C07263=1105.000,381.902,-90.712,-179.506,16.988,151.525
C07264=1105.007,382.149,-90.748,-179.503,16.992,151.526
C07265=1105.012,382.396,-90.785,-179.501,16.996,151.526
C07266=1105.019,382.643,-90.822,-179.498,17.001,151.527
C07267=1105.028,383.057,-90.883,-179.494,17.008,151.528
C07268=1105.037,383.470,-90.944,-179.490,17.016,151.529
C07269=1105.047,383.884,-91.005,-179.484,17.024,151.530
C07270=1105.056,384.298,-91.066,-179.480,17.032,151.531
C07271=1105.061,384.545,-91.103,-179.478,17.037,151.532
C07272=1105.067,384.792,-91.140,-179.476,17.041,151.532
C07273=1105.073,385.040,-91.177,-179.473,17.046,151.533
C07274=1105.078,385.286,-91.213,-179.470,17.051,151.534
C07275=1105.084,385.533,-91.250,-179.468,17.056,151.534
C07276=1105.090,385.781,-91.287,-179.465,17.060,151.535
C07277=1105.096,386.028,-91.323,-179.462,17.065,151.536
C07278=1105.101,386.274,-91.360,-179.460,17.070,151.536
C07279=1105.106,386.522,-91.397,-179.457,17.075,151.537
C07280=1105.112,386.769,-91.434,-179.454,17.080,151.538
C07281=1105.118,387.016,-91.471,-179.453,17.084,151.538
C07282=1105.124,387.264,-91.508,-179.450,17.089,151.539
C07283=1105.129,387.510,-91.544,-179.447,17.094,151.540
C07284=1105.135,387.758,-91.581,-179.445,17.098,151.540
C07285=1105.141,388.005,-91.618,-179.442,17.104,151.541
C07286=1105.147,388.251,-91.656,-179.440,17.108,151.542
C07287=1105.152,388.499,-91.693,-179.437,17.113,151.543
C07288=1105.158,388.746,-91.730,-179.435,17.118,151.543
C07289=1105.163,388.993,-91.766,-179.432,17.123,151.544
C07290=1105.169,389.240,-91.803,-179.429,17.128,151.545
C07291=1105.175,389.487,-91.840,-179.427,17.133,151.546
C07292=1105.181,389.734,-91.878,-179.424,17.138,151.546
C07293=1105.186,389.981,-91.915,-179.422,17.143,151.547
C07294=1105.192,390.229,-91.952,-179.419,17.148,151.548
C07295=1105.198,390.476,-91.988,-179.417,17.153,151.548
C07296=1105.204,390.722,-92.026,-179.414,17.158,151.549
C07297=1105.210,390.970,-92.063,-179.412,17.164,151.550
C07298=1105.216,391.217,-92.100,-179.409,17.168,151.551
C07299=1105.221,391.463,-92.137,-179.407,17.174,151.552
C07300=1105.226,391.711,-92.174,-179.404,17.179,151.552
C07301=1105.232,391.958,-92.211,-179.402,17.184,151.553
C07302=1105.238,392.205,-92.249,-179.399,17.189,151.554
C07303=1105.244,392.452,-92.286,-179.397,17.194,151.555
C07304=1105.249,392.699,-92.324,-179.394,17.199,151.555
C07305=1105.255,392.946,-92.361,-179.392,17.204,151.556
C07306=1105.261,393.194,-92.398,-179.390,17.210,151.557
C07307=1105.267,393.440,-92.436,-179.387,17.215,151.558
C07308=1105.272,393.688,-92.473,-179.385,17.220,151.559
C07309=1105.278,393.934,-92.511,-179.383,17.225,151.560
C07310=1105.284,394.182,-92.548,-179.380,17.231,151.560
C07311=1105.290,394.428,-92.585,-179.378,17.236,151.561
C07312=1105.295,394.676,-92.622,-179.376,17.241,151.562
C07313=1105.301,394.923,-92.660,-179.373,17.247,151.563
C07314=1105.307,395.170,-92.697,-179.371,17.252,151.564
C07315=1105.313,395.417,-92.735,-179.369,17.257,151.565
C07316=1105.318,395.664,-92.772,-179.366,17.263,151.566
C07317=1105.323,395.911,-92.810,-179.364,17.268,151.567
C07318=1105.329,396.158,-92.848,-179.361,17.274,151.567
C07319=1105.334,396.371,-92.881,-179.359,17.278,151.568
C07320=1105.339,396.584,-92.913,-179.358,17.283,151.569
C07321=1105.344,396.797,-92.945,-179.355,17.288,151.570
C07322=1105.349,397.009,-92.977,-179.354,17.293,151.571
C07323=1105.354,397.223,-93.010,-179.351,17.298,151.571
C07324=1105.359,397.435,-93.042,-179.350,17.302,151.572
C07325=1105.364,397.648,-93.075,-179.348,17.307,151.573
C07326=1105.369,397.861,-93.108,-179.345,17.312,151.574
C07327=1105.375,398.108,-93.145,-179.343,17.317,151.575
C07328=1105.380,398.355,-93.182,-179.341,17.323,151.576
C07329=1105.385,398.602,-93.221,-179.339,17.328,151.577
C07330=1105.391,398.849,-93.259,-179.337,17.334,151.578
C07331=1105.397,399.096,-93.296,-179.334,17.340,151.579
C07332=1105.403,399.344,-93.334,-179.332,17.346,151.580
C07333=1105.408,399.591,-93.372,-179.329,17.351,151.580
C07334=1105.414,399.838,-93.410,-179.327,17.357,151.581
C07335=1105.420,400.085,-93.448,-179.325,17.363,151.582
C07336=1105.425,400.331,-93.486,-179.322,17.369,151.584
C07337=1105.431,400.578,-93.524,-179.320,17.375,151.585
C07338=1105.436,400.825,-93.562,-179.318,17.380,151.585
C07339=1105.442,401.072,-93.600,-179.316,17.386,151.587
C07340=1105.448,401.320,-93.638,-179.313,17.392,151.588
C07341=1105.454,401.567,-93.676,-179.311,17.398,151.589
C07342=1105.460,401.814,-93.713,-179.309,17.404,151.590
C07343=1105.465,402.061,-93.752,-179.307,17.409,151.591
C07344=1105.471,402.308,-93.789,-179.305,17.416,151.592
C07345=1105.476,402.555,-93.828,-179.302,17.422,151.593
C07346=1105.482,402.802,-93.866,-179.300,17.428,151.594
C07347=1105.488,403.049,-93.904,-179.299,17.434,151.595
C07348=1105.493,403.296,-93.942,-179.296,17.440,151.596
C07349=1105.499,403.542,-93.981,-179.294,17.446,151.597
C07350=1105.505,403.790,-94.019,-179.292,17.452,151.598
C07351=1105.511,404.037,-94.058,-179.289,17.458,151.599
C07352=1105.517,404.284,-94.095,-179.287,17.464,151.600
C07353=1105.522,404.531,-94.134,-179.285,17.470,151.601
C07354=1105.528,404.778,-94.172,-179.283,17.476,151.603
C07355=1105.533,405.025,-94.210,-179.281,17.482,151.604
C07356=1105.539,405.272,-94.248,-179.279,17.488,151.605
C07357=1105.545,405.518,-94.287,-179.276,17.495,151.606
C07358=1105.551,405.766,-94.325,-179.274,17.501,151.607
C07359=1105.556,406.013,-94.363,-179.272,17.508,151.608
C07360=1105.562,406.260,-94.402,-179.270,17.514,151.609
C07361=1105.568,406.506,-94.440,-179.268,17.520,151.611
C07362=1105.574,406.754,-94.479,-179.266,17.527,151.612
C07363=1105.579,407.001,-94.517,-179.264,17.532,151.613
C07364=1105.585,407.247,-94.556,-179.261,17.539,151.614
C07365=1105.591,407.495,-94.594,-179.259,17.545,151.615
C07366=1105.596,407.742,-94.633,-179.258,17.552,151.617
C07367=1105.602,407.988,-94.671,-179.255,17.558,151.618
C07368=1105.607,408.235,-94.710,-179.254,17.565,151.619
C07369=1105.613,408.483,-94.748,-179.251,17.572,151.620
C07370=1105.618,408.729,-94.787,-179.249,17.578,151.621
C07371=1105.624,408.976,-94.826,-179.247,17.584,151.623
C07372=1105.630,409.223,-94.865,-179.245,17.591,151.624
C07373=1105.636,409.470,-94.903,-179.243,17.598,151.625
C07374=1105.641,409.716,-94.942,-179.241,17.604,151.626
C07375=1105.646,409.930,-94.975,-179.239,17.610,151.628
C07376=1105.650,410.142,-95.008,-179.237,17.616,151.629
C07377=1105.656,410.355,-95.042,-179.235,17.622,151.630
C07378=1105.661,410.568,-95.076,-179.234,17.627,151.631
C07379=1105.665,410.780,-95.109,-179.232,17.633,151.632
C07380=1105.670,410.994,-95.143,-179.230,17.639,151.633
C07381=1105.675,411.206,-95.176,-179.229,17.645,151.634
C07382=1105.680,411.419,-95.209,-179.227,17.651,151.635
C07383=1105.686,411.665,-95.248,-179.225,17.657,151.637
C07384=1105.692,411.913,-95.287,-179.223,17.664,151.638
C07385=1105.697,412.159,-95.326,-179.221,17.671,151.639
C07386=1105.703,412.406,-95.365,-179.219,17.678,151.641
C07387=1105.709,412.653,-95.404,-179.217,17.685,151.642
C07388=1105.714,412.900,-95.443,-179.215,17.692,151.643
C07389=1105.720,413.147,-95.482,-179.213,17.699,151.645
C07390=1105.725,413.394,-95.520,-179.210,17.706,151.646
C07391=1105.731,413.641,-95.560,-179.209,17.713,151.647
C07392=1105.737,413.888,-95.599,-179.207,17.720,151.649
C07393=1105.742,414.134,-95.638,-179.205,17.726,151.650
C07394=1105.748,414.381,-95.677,-179.203,17.734,151.652
C07395=1105.754,414.628,-95.715,-179.201,17.741,151.653
C07396=1105.760,414.875,-95.755,-179.199,17.748,151.654
C07397=1105.766,415.121,-95.794,-179.197,17.755,151.656
C07398=1105.772,415.369,-95.833,-179.195,17.762,151.657
C07399=1105.777,415.615,-95.872,-179.193,17.770,151.659
C07400=1105.783,415.862,-95.912,-179.192,17.776,151.660
C07401=1105.789,416.109,-95.951,-179.189,17.784,151.662
C07402=1105.795,416.356,-95.990,-179.187,17.791,151.663
C07403=1105.800,416.602,-96.029,-179.185,17.799,151.665
C07404=1105.806,416.850,-96.069,-179.184,17.805,151.666
C07405=1105.811,417.096,-96.108,-179.182,17.813,151.667
C07406=1105.817,417.343,-96.148,-179.180,17.820,151.669
C07407=1105.823,417.590,-96.187,-179.178,17.828,151.671
C07408=1105.829,417.837,-96.226,-179.176,17.835,151.672
C07409=1105.834,418.083,-96.265,-179.175,17.843,151.674
C07410=1105.840,418.331,-96.305,-179.173,17.850,151.675
C07411=1105.845,418.577,-96.344,-179.171,17.858,151.677
C07412=1105.851,418.824,-96.384,-179.169,17.865,151.678
C07413=1105.857,419.071,-96.423,-179.167,17.873,151.680
C07414=1105.863,419.318,-96.462,-179.165,17.881,151.681
C07415=1105.868,419.564,-96.503,-179.164,17.888,151.683
C07416=1105.874,419.811,-96.542,-179.162,17.895,151.684
C07417=1105.880,420.058,-96.581,-179.160,17.903,151.686
C07418=1105.885,420.305,-96.621,-179.158,17.911,151.688
C07419=1105.891,420.551,-96.661,-179.156,17.919,151.689
C07420=1105.897,420.798,-96.700,-179.154,17.927,151.691
C07421=1105.903,421.045,-96.740,-179.152,17.934,151.693
C07422=1105.907,421.292,-96.779,-179.151,17.942,151.694
C07423=1105.914,421.538,-96.820,-179.149,17.950,151.696
C07424=1105.920,421.785,-96.859,-179.147,17.958,151.698
C07425=1105.926,422.031,-96.899,-179.146,17.965,151.699
C07426=1105.931,422.279,-96.939,-179.144,17.973,151.701
C07427=1105.937,422.526,-96.978,-179.143,17.982,151.703
C07428=1105.943,422.772,-97.018,-179.141,17.989,151.704
C07429=1105.948,423.019,-97.058,-179.139,17.997,151.706
C07430=1105.954,423.265,-97.098,-179.137,18.005,151.708
C07431=1105.958,423.484,-97.133,-179.135,18.013,151.709
C07432=1105.964,423.704,-97.168,-179.134,18.020,151.711
C07433=1105.969,423.923,-97.205,-179.133,18.027,151.712
C07434=1105.974,424.143,-97.240,-179.131,18.035,151.714
C07435=1105.979,424.362,-97.275,-179.130,18.042,151.715
C07436=1105.984,424.581,-97.311,-179.128,18.050,151.717
C07437=1105.989,424.800,-97.346,-179.127,18.057,151.719
C07438=1105.994,425.020,-97.381,-179.126,18.064,151.720
C07439=1106.000,425.267,-97.422,-179.124,18.072,151.722
C07440=1106.005,425.512,-97.462,-179.122,18.080,151.724
C07441=1106.011,425.760,-97.502,-179.121,18.088,151.725
C07442=1106.017,426.006,-97.542,-179.119,18.098,151.727
C07443=1106.022,426.252,-97.582,-179.117,18.106,151.729
C07444=1106.028,426.500,-97.622,-179.115,18.114,151.731
C07445=1106.034,426.746,-97.663,-179.114,18.123,151.733
C07446=1106.040,426.993,-97.703,-179.112,18.131,151.735
C07447=1106.045,427.239,-97.743,-179.111,18.139,151.737
C07448=1106.051,427.486,-97.783,-179.110,18.148,151.738
C07449=1106.057,427.733,-97.823,-179.108,18.156,151.740
C07450=1106.062,427.979,-97.864,-179.106,18.165,151.742
C07451=1106.068,428.226,-97.904,-179.104,18.174,151.744
C07452=1106.074,428.472,-97.944,-179.103,18.183,151.746
C07453=1106.079,428.720,-97.985,-179.102,18.191,151.748
C07454=1106.085,428.966,-98.024,-179.100,18.200,151.750
C07455=1106.091,429.213,-98.065,-179.099,18.209,151.752
C07456=1106.097,429.459,-98.106,-179.097,18.218,151.754
C07457=1106.103,429.706,-98.146,-179.096,18.226,151.756
C07458=1106.108,429.952,-98.186,-179.094,18.235,151.758
C07459=1106.114,430.199,-98.227,-179.093,18.244,151.760
C07460=1106.120,430.445,-98.267,-179.091,18.254,151.762
C07461=1106.125,430.691,-98.308,-179.090,18.262,151.764
C07462=1106.131,430.938,-98.348,-179.089,18.271,151.766
C07463=1106.136,431.185,-98.389,-179.088,18.280,151.768
C07464=1106.142,431.432,-98.430,-179.086,18.290,151.770
C07465=1106.148,431.678,-98.470,-179.084,18.298,151.772
C07466=1106.153,431.925,-98.510,-179.083,18.308,151.774
C07467=1106.159,432.171,-98.551,-179.081,18.317,151.776
C07468=1106.165,432.418,-98.593,-179.080,18.326,151.778
C07469=1106.171,432.664,-98.633,-179.079,18.335,151.780
C07470=1106.177,432.911,-98.673,-179.077,18.345,151.782
C07471=1106.182,433.157,-98.714,-179.076,18.354,151.784
C07472=1106.188,433.404,-98.755,-179.075,18.363,151.787
C07473=1106.194,433.650,-98.796,-179.073,18.373,151.789
C07474=1106.199,433.897,-98.837,-179.072,18.382,151.791
C07475=1106.205,434.144,-98.877,-179.071,18.391,151.793
C07476=1106.210,434.390,-98.918,-179.070,18.401,151.795
C07477=1106.216,434.636,-98.959,-179.069,18.410,151.797
C07478=1106.222,434.883,-99.000,-179.067,18.421,151.800
C07479=1106.227,435.130,-99.041,-179.066,18.430,151.802
C07480=1106.233,435.376,-99.082,-179.065,18.439,151.804
C07481=1106.238,435.622,-99.123,-179.064,18.449,151.806
C07482=1106.244,435.868,-99.164,-179.063,18.459,151.809
C07483=1106.250,436.115,-99.205,-179.061,18.469,151.811
C07484=1106.255,436.362,-99.246,-179.060,18.478,151.813
C07485=1106.261,436.608,-99.287,-179.059,18.488,151.815
C07486=1106.267,436.855,-99.328,-179.058,18.498,151.818
C07487=1106.272,437.072,-99.364,-179.057,18.507,151.820
C07488=1106.277,437.290,-99.400,-179.056,18.516,151.822
C07489=1106.282,437.508,-99.437,-179.055,18.524,151.824
C07490=1106.287,437.726,-99.474,-179.054,18.533,151.826
C07491=1106.292,437.944,-99.510,-179.053,18.542,151.828
C07492=1106.297,438.162,-99.546,-179.052,18.551,151.830
C07493=1106.302,438.380,-99.582,-179.051,18.560,151.832
C07494=1106.307,438.598,-99.619,-179.050,18.569,151.834
C07495=1106.313,438.844,-99.660,-179.049,18.579,151.837
C07496=1106.318,439.091,-99.701,-179.048,18.589,151.839
C07497=1106.324,439.337,-99.743,-179.047,18.600,151.842
C07498=1106.330,439.583,-99.784,-179.046,18.609,151.844
C07499=1106.336,439.829,-99.825,-179.045,18.620,151.846
C07500=1106.341,440.076,-99.867,-179.044,18.630,151.849
C07501=1106.347,440.323,-99.908,-179.043,18.641,151.851
C07502=1106.353,440.569,-99.950,-179.041,18.651,151.854
C07503=1106.359,440.815,-99.991,-179.041,18.661,151.856
C07504=1106.365,441.062,-100.032,-179.040,18.672,151.859
C07505=1106.370,441.308,-100.074,-179.039,18.682,151.861
C07506=1106.376,441.555,-100.115,-179.038,18.693,151.864
C07507=1106.382,441.801,-100.157,-179.037,18.704,151.866
C07508=1106.388,442.047,-100.198,-179.037,18.714,151.869
C07509=1106.393,442.293,-100.240,-179.036,18.725,151.872
C07510=1106.399,442.540,-100.282,-179.034,18.736,151.874
C07511=1106.405,442.786,-100.323,-179.034,18.747,151.877
C07512=1106.410,443.032,-100.365,-179.033,18.758,151.879
C07513=1106.416,443.279,-100.407,-179.032,18.769,151.882
C07514=1106.421,443.525,-100.449,-179.032,18.779,151.885
C07515=1106.427,443.771,-100.490,-179.031,18.790,151.887
C07516=1106.433,444.018,-100.532,-179.030,18.801,151.890
C07517=1106.438,444.264,-100.574,-179.030,18.812,151.893
C07518=1106.444,444.510,-100.615,-179.029,18.823,151.895
C07519=1106.449,444.757,-100.657,-179.029,18.834,151.898
C07520=1106.455,445.003,-100.699,-179.029,18.845,151.901
C07521=1106.461,445.249,-100.741,-179.030,18.855,151.904
C07522=1106.467,445.496,-100.782,-179.030,18.866,151.907
C07523=1106.472,445.742,-100.824,-179.030,18.877,151.909
C07524=1106.478,445.988,-100.866,-179.031,18.887,151.912
C07525=1106.483,446.234,-100.909,-179.032,18.898,151.915
C07526=1106.489,446.480,-100.950,-179.032,18.909,151.918
C07527=1106.494,446.727,-100.992,-179.033,18.920,151.921
C07528=1106.501,446.974,-101.034,-179.034,18.930,151.924
C07529=1106.506,447.220,-101.076,-179.035,18.941,151.927
C07530=1106.512,447.467,-101.117,-179.036,18.952,151.930
C07531=1106.518,447.713,-101.160,-179.037,18.963,151.933
C07532=1106.523,447.959,-101.202,-179.039,18.973,151.936
C07533=1106.529,448.205,-101.244,-179.040,18.984,151.939
C07534=1106.534,448.452,-101.286,-179.042,18.994,151.942
C07535=1106.539,448.698,-101.329,-179.043,19.005,151.945
C07536=1106.546,448.945,-101.370,-179.045,19.015,151.948
C07537=1106.551,449.191,-101.412,-179.047,19.026,151.951
C07538=1106.558,449.437,-101.455,-179.049,19.037,151.954
C07539=1106.563,449.683,-101.497,-179.050,19.047,151.957
C07540=1106.568,449.930,-101.539,-179.053,19.058,151.960
C07541=1106.574,450.175,-101.581,-179.054,19.068,151.963
C07542=1106.579,450.422,-101.623,-179.057,19.079,151.966
C07543=1106.174,450.414,-101.743,-179.136,19.309,152.039
C07544=1106.168,450.169,-101.701,-179.134,19.299,152.036
C07545=1106.162,449.922,-101.659,-179.132,19.288,152.033
C07546=1106.157,449.676,-101.616,-179.130,19.277,152.030
C07547=1106.151,449.430,-101.575,-179.128,19.267,152.027
C07548=1106.145,449.183,-101.532,-179.126,19.256,152.024
C07549=1106.140,448.937,-101.490,-179.125,19.245,152.021
C07550=1106.134,448.691,-101.448,-179.123,19.235,152.018
C07551=1106.129,448.444,-101.406,-179.121,19.224,152.015
C07552=1106.123,448.198,-101.363,-179.120,19.213,152.012
C07553=1106.116,447.952,-101.322,-179.118,19.203,152.009
C07554=1106.111,447.705,-101.280,-179.117,19.192,152.006
C07555=1106.105,447.459,-101.237,-179.116,19.181,152.003
C07556=1106.100,447.213,-101.195,-179.115,19.170,152.000
C07557=1106.095,446.966,-101.153,-179.114,19.160,151.997
C07558=1106.089,446.720,-101.112,-179.113,19.149,151.994
C07559=1106.083,446.474,-101.069,-179.112,19.138,151.991
C07560=1106.077,446.228,-101.028,-179.112,19.127,151.988
C07561=1106.071,445.981,-100.985,-179.112,19.116,151.986
C07562=1106.066,445.734,-100.943,-179.111,19.106,151.983
C07563=1106.060,445.489,-100.901,-179.111,19.095,151.980
C07564=1106.055,445.242,-100.859,-179.110,19.084,151.977
C07565=1106.049,444.996,-100.817,-179.110,19.073,151.974
C07566=1106.043,444.750,-100.776,-179.110,19.062,151.971
C07567=1106.038,444.503,-100.734,-179.110,19.051,151.969
C07568=1106.032,444.257,-100.692,-179.110,19.040,151.966
C07569=1106.026,444.011,-100.650,-179.111,19.029,151.963
C07570=1106.020,443.765,-100.608,-179.112,19.018,151.960
C07571=1106.015,443.519,-100.566,-179.112,19.008,151.958
C07572=1106.009,443.272,-100.525,-179.113,18.996,151.955
C07573=1106.004,443.026,-100.483,-179.114,18.985,151.952
C07574=1105.998,442.780,-100.441,-179.115,18.974,151.950
C07575=1105.992,442.533,-100.400,-179.115,18.964,151.947
C07576=1105.987,442.287,-100.358,-179.117,18.953,151.945
C07577=1105.980,442.040,-100.316,-179.118,18.942,151.942
C07578=1105.975,441.795,-100.275,-179.118,18.931,151.939
C07579=1105.969,441.548,-100.233,-179.119,18.920,151.937
C07580=1105.964,441.301,-100.192,-179.121,18.909,151.934
C07581=1105.958,441.055,-100.151,-179.121,18.899,151.932
C07582=1105.952,440.809,-100.109,-179.122,18.888,151.929
C07583=1105.947,440.562,-100.067,-179.123,18.878,151.927
C07584=1105.941,440.316,-100.026,-179.124,18.867,151.924
C07585=1105.935,440.070,-99.984,-179.126,18.857,151.922
C07586=1105.929,439.824,-99.943,-179.126,18.847,151.919
C07587=1105.923,439.577,-99.902,-179.127,18.836,151.917
C07588=1105.917,439.331,-99.860,-179.128,18.826,151.914
C07589=1105.912,439.084,-99.818,-179.130,18.815,151.912
C07590=1105.906,438.838,-99.777,-179.131,18.805,151.910
C07591=1105.901,438.591,-99.736,-179.132,18.795,151.907
C07592=1105.896,438.375,-99.700,-179.133,18.786,151.905
C07593=1105.890,438.159,-99.664,-179.134,18.777,151.903
C07594=1105.885,437.943,-99.627,-179.135,18.768,151.901
C07595=1105.880,437.727,-99.591,-179.136,18.759,151.899
C07596=1105.875,437.512,-99.556,-179.137,18.750,151.897
C07597=1105.870,437.297,-99.520,-179.138,18.742,151.895
C07598=1105.865,437.081,-99.483,-179.139,18.733,151.893
C07599=1105.860,436.865,-99.447,-179.140,18.724,151.891
C07600=1105.854,436.618,-99.406,-179.141,18.714,151.888
C07601=1105.848,436.372,-99.365,-179.143,18.704,151.886
C07602=1105.843,436.126,-99.325,-179.143,18.695,151.884
C07603=1105.837,435.879,-99.283,-179.145,18.684,151.881
C07604=1105.832,435.633,-99.242,-179.146,18.675,151.879
C07605=1105.826,435.386,-99.201,-179.148,18.665,151.877
C07606=1105.820,435.140,-99.160,-179.149,18.655,151.875
C07607=1105.814,434.893,-99.119,-179.150,18.646,151.872
C07608=1105.809,434.647,-99.078,-179.151,18.636,151.870
C07609=1105.804,434.400,-99.038,-179.152,18.626,151.868
C07610=1105.798,434.154,-98.996,-179.154,18.616,151.866
C07611=1105.792,433.907,-98.955,-179.155,18.607,151.864
C07612=1105.786,433.661,-98.915,-179.157,18.597,151.861
C07613=1105.780,433.414,-98.873,-179.158,18.588,151.859
C07614=1105.775,433.168,-98.833,-179.159,18.579,151.857
C07615=1105.770,432.921,-98.792,-179.161,18.569,151.855
C07616=1105.764,432.675,-98.751,-179.162,18.560,151.853
C07617=1105.758,432.428,-98.710,-179.163,18.550,151.851
C07618=1105.752,432.182,-98.670,-179.165,18.541,151.849
C07619=1105.747,431.936,-98.629,-179.166,18.532,151.847
C07620=1105.741,431.689,-98.589,-179.167,18.523,151.845
C07621=1105.735,431.442,-98.548,-179.169,18.513,151.842
C07622=1105.730,431.195,-98.507,-179.171,18.504,151.840
C07623=1105.723,430.949,-98.466,-179.172,18.495,151.838
C07624=1105.718,430.703,-98.426,-179.173,18.486,151.836
C07625=1105.712,430.456,-98.385,-179.175,18.477,151.834
C07626=1105.707,430.210,-98.344,-179.176,18.468,151.832
C07627=1105.701,429.963,-98.304,-179.178,18.459,151.830
C07628=1105.695,429.717,-98.264,-179.179,18.450,151.828
C07629=1105.690,429.470,-98.223,-179.181,18.441,151.826
C07630=1105.684,429.223,-98.182,-179.182,18.432,151.824
C07631=1105.678,428.977,-98.142,-179.183,18.423,151.822
C07632=1105.672,428.730,-98.102,-179.185,18.415,151.820
C07633=1105.667,428.484,-98.061,-179.187,18.405,151.818
C07634=1105.661,428.237,-98.022,-179.189,18.397,151.816
C07635=1105.655,427.990,-97.981,-179.190,18.388,151.814
C07636=1105.649,427.743,-97.941,-179.191,18.380,151.813
C07637=1105.644,427.497,-97.900,-179.193,18.371,151.811
C07638=1105.638,427.250,-97.860,-179.195,18.363,151.809
C07639=1105.632,427.004,-97.820,-179.197,18.353,151.807
C07640=1105.627,426.757,-97.780,-179.198,18.345,151.805
C07641=1105.621,426.511,-97.740,-179.200,18.336,151.803
C07642=1105.615,426.264,-97.699,-179.201,18.328,151.801
C07643=1105.609,426.017,-97.659,-179.203,18.319,151.800
C07644=1105.604,425.771,-97.619,-179.204,18.311,151.798
C07645=1105.598,425.524,-97.578,-179.206,18.303,151.796
C07646=1105.592,425.277,-97.538,-179.207,18.294,151.794
C07647=1105.587,425.031,-97.499,-179.209,18.286,151.792
C07648=1105.581,424.811,-97.463,-179.211,18.278,151.791
C07649=1105.576,424.592,-97.427,-179.212,18.271,151.789
C07650=1105.572,424.372,-97.392,-179.214,18.264,151.788
C07651=1105.567,424.153,-97.356,-179.215,18.256,151.786
C07652=1105.561,423.933,-97.321,-179.216,18.249,151.784
C07653=1105.556,423.714,-97.285,-179.219,18.241,151.783
C07654=1105.552,423.494,-97.250,-179.220,18.234,151.781
C07655=1105.547,423.275,-97.214,-179.222,18.227,151.780
C07656=1105.541,423.028,-97.174,-179.224,18.219,151.778
C07657=1105.534,422.782,-97.134,-179.225,18.211,151.776
C07658=1105.530,422.535,-97.094,-179.227,18.202,151.775
C07659=1105.523,422.288,-97.054,-179.229,18.194,151.773
C07660=1105.517,422.041,-97.015,-179.230,18.187,151.771
C07661=1105.512,421.795,-96.975,-179.232,18.179,151.770
C07662=1105.506,421.548,-96.935,-179.233,18.171,151.768
C07663=1105.500,421.301,-96.895,-179.235,18.163,151.766
C07664=1105.495,421.054,-96.856,-179.237,18.155,151.765
C07665=1105.489,420.808,-96.816,-179.239,18.147,151.763
C07666=1105.483,420.561,-96.777,-179.241,18.140,151.761
C07667=1105.477,420.314,-96.737,-179.243,18.132,151.760
C07668=1105.472,420.067,-96.696,-179.245,18.124,151.758
C07669=1105.466,419.821,-96.657,-179.247,18.116,151.756
C07670=1105.460,419.574,-96.618,-179.248,18.108,151.755
C07671=1105.455,419.327,-96.579,-179.250,18.100,151.753
C07672=1105.449,419.080,-96.538,-179.252,18.093,151.752
C07673=1105.444,418.834,-96.499,-179.254,18.086,151.750
C07674=1105.438,418.587,-96.460,-179.256,18.078,151.749
C07675=1105.432,418.340,-96.421,-179.258,18.070,151.747
C07676=1105.427,418.093,-96.381,-179.260,18.062,151.745
C07677=1105.421,417.847,-96.341,-179.262,18.055,151.744
C07678=1105.415,417.599,-96.302,-179.263,18.047,151.742
C07679=1105.409,417.354,-96.262,-179.265,18.040,151.741
C07680=1105.403,417.106,-96.223,-179.267,18.033,151.739
C07681=1105.399,416.860,-96.183,-179.269,18.025,151.738
C07682=1105.392,416.613,-96.144,-179.271,18.017,151.736
C07683=1105.387,416.366,-96.105,-179.273,18.010,151.735
C07684=1105.381,416.119,-96.065,-179.275,18.003,151.733
C07685=1105.375,415.872,-96.026,-179.277,17.996,151.732
C07686=1105.369,415.625,-95.987,-179.279,17.988,151.730
C07687=1105.363,415.378,-95.947,-179.281,17.981,151.729
C07688=1105.358,415.131,-95.909,-179.282,17.974,151.728
C07689=1105.352,414.884,-95.870,-179.285,17.967,151.726
C07690=1105.347,414.638,-95.830,-179.287,17.960,151.725
C07691=1105.341,414.391,-95.791,-179.288,17.953,151.723
C07692=1105.335,414.144,-95.752,-179.291,17.946,151.722
C07693=1105.330,413.898,-95.713,-179.293,17.938,151.720
C07694=1105.324,413.651,-95.673,-179.294,17.932,151.719
C07695=1105.318,413.403,-95.635,-179.296,17.924,151.718
C07696=1105.312,413.157,-95.596,-179.299,17.917,151.716
C07697=1105.306,412.910,-95.557,-179.300,17.910,151.715
C07698=1105.300,412.663,-95.518,-179.303,17.903,151.714
C07699=1105.295,412.416,-95.479,-179.305,17.896,151.712
C07700=1105.289,412.169,-95.440,-179.306,17.889,151.711
C07701=1105.283,411.922,-95.401,-179.309,17.882,151.709
C07702=1105.278,411.675,-95.363,-179.311,17.875,151.708
C07703=1105.272,411.428,-95.323,-179.313,17.869,151.707
C07704=1105.267,411.215,-95.290,-179.314,17.862,151.706
C07705=1105.262,411.003,-95.256,-179.316,17.857,151.704
C07706=1105.257,410.790,-95.223,-179.318,17.851,151.703
C07707=1105.252,410.577,-95.189,-179.319,17.845,151.702
C07708=1105.248,410.365,-95.155,-179.321,17.839,151.701
C07709=1105.243,410.151,-95.123,-179.323,17.833,151.700
C07710=1105.238,409.938,-95.089,-179.325,17.828,151.699
C07711=1105.233,409.725,-95.055,-179.327,17.821,151.698
C07712=1105.227,409.479,-95.016,-179.329,17.815,151.696
C07713=1105.222,409.232,-94.978,-179.331,17.808,151.695
C07714=1105.216,408.984,-94.939,-179.333,17.802,151.694
C07715=1105.210,408.738,-94.901,-179.335,17.795,151.693
C07716=1105.205,408.491,-94.862,-179.337,17.788,151.691
C07717=1105.199,408.244,-94.823,-179.339,17.781,151.690
C07718=1105.194,407.996,-94.785,-179.341,17.776,151.689
C07719=1105.187,407.750,-94.746,-179.344,17.769,151.688
C07720=1105.182,407.503,-94.708,-179.346,17.762,151.686
C07721=1105.177,407.256,-94.669,-179.348,17.755,151.685
C07722=1105.170,407.009,-94.631,-179.350,17.749,151.684
C07723=1105.165,406.762,-94.592,-179.352,17.743,151.683
C07724=1105.159,406.515,-94.553,-179.354,17.737,151.682
C07725=1105.154,406.268,-94.514,-179.356,17.730,151.680
C07726=1105.148,406.021,-94.477,-179.359,17.724,151.679
C07727=1105.142,405.774,-94.438,-179.360,17.717,151.678
C07728=1105.136,405.527,-94.400,-179.362,17.711,151.677
C07729=1105.131,405.280,-94.361,-179.365,17.705,151.676
C07730=1105.126,405.033,-94.323,-179.367,17.699,151.675
C07731=1105.119,404.786,-94.285,-179.369,17.692,151.674
C07732=1105.114,404.539,-94.246,-179.371,17.686,151.672
C07733=1105.108,404.292,-94.209,-179.373,17.680,151.671
C07734=1105.103,404.046,-94.169,-179.376,17.674,151.670
C07735=1105.096,403.798,-94.131,-179.378,17.668,151.669
C07736=1105.091,403.551,-94.093,-179.380,17.662,151.668
C07737=1105.085,403.305,-94.055,-179.383,17.655,151.667
C07738=1105.080,403.057,-94.017,-179.385,17.650,151.666
C07739=1105.073,402.810,-93.979,-179.387,17.644,151.665
C07740=1105.068,402.563,-93.940,-179.389,17.637,151.664
C07741=1105.062,402.316,-93.903,-179.391,17.631,151.663
C07742=1105.057,402.069,-93.864,-179.393,17.625,151.661
C07743=1105.051,401.822,-93.827,-179.395,17.620,151.661
C07744=1105.045,401.575,-93.788,-179.398,17.613,151.659
C07745=1105.040,401.328,-93.750,-179.400,17.608,151.658
C07746=1105.034,401.081,-93.712,-179.402,17.602,151.657
C07747=1105.029,400.834,-93.674,-179.404,17.596,151.656
C07748=1105.023,400.587,-93.636,-179.407,17.589,151.655
C07749=1105.017,400.340,-93.598,-179.409,17.584,151.654
C07750=1105.011,400.093,-93.560,-179.411,17.578,151.653
C07751=1105.005,399.846,-93.522,-179.414,17.572,151.652
C07752=1105.000,399.599,-93.484,-179.416,17.566,151.651
C07753=1104.994,399.352,-93.447,-179.418,17.560,151.650
C07754=1104.988,399.105,-93.409,-179.421,17.555,151.649
C07755=1104.983,398.858,-93.371,-179.423,17.549,151.648
C07756=1104.977,398.611,-93.333,-179.425,17.544,151.647
C07757=1104.971,398.364,-93.295,-179.428,17.537,151.646
C07758=1104.965,398.116,-93.258,-179.430,17.532,151.645
C07759=1104.960,397.869,-93.219,-179.432,17.526,151.644
C07760=1104.955,397.657,-93.187,-179.434,17.522,151.644
C07761=1104.950,397.443,-93.154,-179.436,17.516,151.643
C07762=1104.945,397.231,-93.121,-179.438,17.512,151.642
C07763=1104.940,397.017,-93.089,-179.440,17.507,151.641
C07764=1104.936,396.805,-93.056,-179.442,17.502,151.640
C07765=1104.931,396.591,-93.024,-179.445,17.497,151.639
C07766=1104.925,396.379,-92.992,-179.446,17.492,151.639
C07767=1104.921,396.166,-92.960,-179.448,17.488,151.638
C07768=1104.915,395.919,-92.921,-179.451,17.482,151.637
C07769=1104.910,395.672,-92.884,-179.453,17.477,151.636
C07770=1104.903,395.424,-92.846,-179.455,17.471,151.635
C07771=1104.898,395.177,-92.809,-179.458,17.466,151.634
C07772=1104.892,394.930,-92.771,-179.460,17.460,151.633
C07773=1104.886,394.683,-92.734,-179.463,17.455,151.633
C07774=1104.880,394.436,-92.697,-179.465,17.450,151.632
C07775=1104.874,394.189,-92.659,-179.467,17.444,151.631
C07776=1104.869,393.942,-92.622,-179.469,17.439,151.630
C07777=1104.864,393.695,-92.584,-179.472,17.434,151.629
C07778=1104.858,393.447,-92.547,-179.474,17.428,151.628
C07779=1104.852,393.201,-92.509,-179.476,17.423,151.627
C07780=1104.847,392.953,-92.472,-179.479,17.418,151.627
C07781=1104.841,392.706,-92.435,-179.481,17.413,151.626
C07782=1104.836,392.460,-92.397,-179.485,17.407,151.625
C07783=1104.830,392.213,-92.360,-179.487,17.402,151.624
C07784=1104.824,391.966,-92.322,-179.490,17.396,151.623
C07785=1104.819,391.718,-92.285,-179.492,17.391,151.623
C07786=1104.812,391.471,-92.249,-179.494,17.386,151.622
C07787=1104.806,391.225,-92.211,-179.497,17.381,151.621
C07788=1104.801,390.977,-92.174,-179.499,17.376,151.620
C07789=1104.795,390.730,-92.137,-179.502,17.371,151.619
C07790=1104.789,390.483,-92.099,-179.504,17.365,151.619
C07791=1104.784,390.236,-92.062,-179.507,17.361,151.618
C07792=1104.778,389.988,-92.025,-179.509,17.355,151.617
C07793=1104.772,389.741,-91.989,-179.512,17.350,151.616
C07794=1104.766,389.495,-91.951,-179.515,17.346,151.616
C07795=1104.760,389.247,-91.914,-179.517,17.340,151.615
C07796=1104.755,389.000,-91.877,-179.519,17.335,151.614
C07797=1104.750,388.753,-91.840,-179.522,17.330,151.613
C07798=1104.744,388.507,-91.803,-179.525,17.325,151.613
C07799=1104.737,388.260,-91.766,-179.527,17.321,151.612
C07800=1104.732,388.012,-91.729,-179.529,17.316,151.611
C07801=1104.726,387.765,-91.692,-179.532,17.311,151.610
C07802=1104.721,387.517,-91.655,-179.534,17.306,151.610
C07803=1104.715,387.271,-91.619,-179.537,17.301,151.609
C07804=1104.709,387.024,-91.582,-179.539,17.296,151.608
C07805=1104.704,386.776,-91.545,-179.542,17.291,151.608
C07806=1104.698,386.529,-91.508,-179.545,17.286,151.607
C07807=1104.691,386.283,-91.471,-179.547,17.281,151.606
C07808=1104.686,386.036,-91.434,-179.550,17.276,151.605
C07809=1104.681,385.789,-91.397,-179.553,17.272,151.605
C07810=1104.675,385.541,-91.360,-179.555,17.267,151.604
C07811=1104.669,385.294,-91.324,-179.558,17.262,151.603
C07812=1104.664,385.046,-91.287,-179.560,17.257,151.603
C07813=1104.659,384.799,-91.251,-179.562,17.253,151.602
C07814=1104.652,384.552,-91.214,-179.565,17.248,151.601
C07815=1104.647,384.305,-91.177,-179.568,17.243,151.601
C07816=1104.637,383.891,-91.116,-179.572,17.235,151.600
C07817=1104.629,383.477,-91.054,-179.577,17.227,151.599
C07818=1104.619,383.063,-90.993,-179.581,17.219,151.598
C07819=1104.609,382.651,-90.931,-179.586,17.212,151.597
C07820=1104.603,382.403,-90.896,-179.589,17.207,151.596
C07821=1104.598,382.155,-90.859,-179.591,17.202,151.595
C07822=1104.591,381.908,-90.822,-179.593,17.198,151.595
C07823=1104.586,381.661,-90.785,-179.596,17.194,151.594
C07824=1104.580,381.414,-90.750,-179.599,17.189,151.594
C07825=1104.575,381.167,-90.713,-179.602,17.184,151.593
C07826=1104.568,380.920,-90.676,-179.605,17.180,151.592
C07827=1104.564,380.672,-90.640,-179.607,17.176,151.592
C07828=1104.557,380.425,-90.604,-179.609,17.171,151.591
C07829=1104.551,380.178,-90.567,-179.612,17.167,151.591
C07830=1104.546,379.930,-90.531,-179.615,17.162,151.590
C07831=1104.540,379.684,-90.495,-179.618,17.158,151.590
C07832=1104.534,379.437,-90.458,-179.620,17.153,151.589
C07833=1104.528,379.189,-90.422,-179.623,17.149,151.589
C07834=1104.523,378.942,-90.386,-179.626,17.145,151.588
C07835=1104.517,378.695,-90.350,-179.629,17.140,151.587
C07836=1104.511,378.447,-90.313,-179.631,17.136,151.587
C07837=1104.506,378.200,-90.277,-179.634,17.132,151.586
C07838=1104.500,377.953,-90.241,-179.637,17.127,151.586
C07839=1104.495,377.706,-90.205,-179.640,17.122,151.585
C07840=1104.489,377.459,-90.169,-179.642,17.119,151.585
C07841=1104.483,377.211,-90.133,-179.645,17.114,151.584
C07842=1104.478,376.964,-90.096,-179.648,17.110,151.584
C07843=1104.472,376.717,-90.060,-179.651,17.105,151.583
C07844=1104.466,376.469,-90.025,-179.653,17.101,151.583
C07845=1104.461,376.222,-89.988,-179.656,17.097,151.582
C07846=1104.455,375.975,-89.952,-179.659,17.093,151.582
C07847=1104.449,375.728,-89.916,-179.661,17.089,151.581
C07848=1104.444,375.480,-89.880,-179.664,17.084,151.581
C07849=1104.438,375.233,-89.845,-179.667,17.080,151.580
C07850=1104.432,374.986,-89.809,-179.670,17.076,151.580
C07851=1104.427,374.738,-89.772,-179.672,17.072,151.579
C07852=1104.421,374.491,-89.736,-179.675,17.067,151.579
C07853=1104.415,374.244,-89.701,-179.678,17.063,151.578
C07854=1104.410,373.997,-89.665,-179.681,17.060,151.578
C07855=1104.404,373.750,-89.629,-179.684,17.055,151.578
C07856=1104.398,373.502,-89.593,-179.687,17.051,151.577
C07857=1104.393,373.255,-89.557,-179.689,17.047,151.577
C07858=1104.387,373.007,-89.521,-179.692,17.043,151.576
C07859=1104.381,372.761,-89.485,-179.695,17.039,151.576
C07860=1104.375,372.513,-89.450,-179.697,17.035,151.575
C07861=1104.370,372.266,-89.414,-179.700,17.031,151.575
C07862=1104.364,372.018,-89.379,-179.704,17.027,151.575
C07863=1104.358,371.771,-89.343,-179.706,17.023,151.574
C07864=1104.353,371.524,-89.307,-179.709,17.019,151.574
C07865=1104.347,371.276,-89.271,-179.711,17.015,151.573
C07866=1104.341,371.029,-89.236,-179.715,17.011,151.573
C07867=1104.335,370.781,-89.200,-179.718,17.007,151.573
C07868=1104.327,370.394,-89.144,-179.722,17.001,151.572
C07869=1104.317,370.008,-89.089,-179.726,16.995,151.571
C07870=1104.309,369.621,-89.034,-179.731,16.989,151.571
C07871=1104.300,369.234,-88.978,-179.736,16.983,151.570
C07872=1104.294,368.986,-88.942,-179.738,16.979,151.570
C07873=1104.289,368.739,-88.906,-179.741,16.975,151.569
C07874=1104.283,368.491,-88.871,-179.744,16.972,151.569
C07875=1104.277,368.244,-88.835,-179.747,16.968,151.569
C07876=1104.271,367.997,-88.800,-179.750,16.964,151.568
C07877=1104.266,367.749,-88.765,-179.753,16.960,151.568
C07878=1104.260,367.502,-88.729,-179.756,16.956,151.568
C07879=1104.255,367.255,-88.694,-179.758,16.952,151.567
C07880=1104.249,367.008,-88.659,-179.762,16.948,151.567
C07881=1104.243,366.760,-88.623,-179.764,16.945,151.567
C07882=1104.238,366.512,-88.588,-179.767,16.941,151.566
C07883=1104.232,366.265,-88.552,-179.771,16.937,151.566
C07884=1104.226,366.018,-88.518,-179.773,16.934,151.566
C07885=1104.220,365.770,-88.482,-179.776,16.930,151.565
C07886=1104.215,365.523,-88.447,-179.779,16.926,151.565
C07887=1104.209,365.276,-88.412,-179.782,16.922,151.565
C07888=1104.203,365.028,-88.376,-179.785,16.919,151.564
C07889=1104.198,364.780,-88.342,-179.788,16.915,151.564
C07890=1104.192,364.533,-88.306,-179.791,16.912,151.564
C07891=1104.186,364.286,-88.271,-179.794,16.908,151.564
C07892=1104.181,364.039,-88.236,-179.796,16.905,151.563
C07893=1104.175,363.791,-88.201,-179.800,16.901,151.563
C07894=1104.170,363.543,-88.166,-179.802,16.898,151.563
C07895=1104.163,363.296,-88.131,-179.806,16.894,151.562
C07896=1104.158,363.048,-88.096,-179.808,16.890,151.562
C07897=1104.152,362.801,-88.061,-179.812,16.887,151.562
C07898=1104.147,362.553,-88.026,-179.814,16.883,151.562
C07899=1104.141,362.306,-87.991,-179.817,16.879,151.561
C07900=1104.135,362.058,-87.956,-179.820,16.876,151.561
C07901=1104.129,361.811,-87.921,-179.823,16.872,151.561
C07902=1104.124,361.564,-87.886,-179.826,16.869,151.561
C07903=1104.118,361.316,-87.851,-179.829,16.865,151.560
C07904=1104.112,361.069,-87.816,-179.832,16.862,151.560
C07905=1104.107,360.822,-87.781,-179.835,16.858,151.560
C07906=1104.101,360.574,-87.746,-179.838,16.855,151.560
C07907=1104.095,360.326,-87.712,-179.841,16.851,151.559
C07908=1104.090,360.079,-87.676,-179.844,16.848,151.559
C07909=1104.084,359.831,-87.642,-179.847,16.845,151.559
C07910=1104.078,359.583,-87.607,-179.850,16.841,151.559
C07911=1104.072,359.337,-87.573,-179.853,16.838,151.558
C07912=1104.067,359.089,-87.538,-179.857,16.835,151.558
C07913=1104.061,358.841,-87.503,-179.859,16.831,151.558
C07914=1104.055,358.594,-87.468,-179.863,16.828,151.558
C07915=1104.050,358.347,-87.434,-179.865,16.825,151.558
C07916=1104.044,358.099,-87.399,-179.869,16.821,151.558
C07917=1104.039,357.851,-87.365,-179.871,16.818,151.557
C07918=1104.032,357.604,-87.330,-179.874,16.815,151.557
C07919=1104.027,357.356,-87.295,-179.878,16.811,151.557
C07920=1104.018,356.984,-87.243,-179.882,16.806,151.557
C07921=1104.010,356.612,-87.191,-179.887,16.802,151.556
C07922=1104.001,356.240,-87.139,-179.892,16.796,151.556
C07923=1103.992,355.868,-87.087,-179.896,16.792,151.556
C07924=1103.987,355.620,-87.053,-179.899,16.788,151.556
C07925=1103.981,355.373,-87.019,-179.902,16.785,151.555
C07926=1103.976,355.125,-86.984,-179.905,16.782,151.555
C07927=1103.970,354.877,-86.950,-179.908,16.778,151.555
C07928=1103.965,354.630,-86.915,-179.911,16.775,151.555
C07929=1103.959,354.382,-86.881,-179.915,16.772,151.555
C07930=1103.953,354.135,-86.847,-179.917,16.769,151.555
C07931=1103.948,353.887,-86.812,-179.920,16.766,151.555
C07932=1103.941,353.639,-86.778,-179.924,16.763,151.554
C07933=1103.936,353.392,-86.743,-179.927,16.760,151.554
C07934=1103.930,353.145,-86.709,-179.929,16.757,151.554
C07935=1103.924,352.897,-86.675,-179.933,16.753,151.554
C07936=1103.919,352.650,-86.640,-179.936,16.750,151.554
C07937=1103.913,352.402,-86.606,-179.939,16.748,151.554
C07938=1103.907,352.154,-86.573,-179.942,16.744,151.554
C07939=1103.902,351.906,-86.538,-179.945,16.741,151.553
C07940=1103.896,351.659,-86.504,-179.948,16.738,151.553
C07941=1103.891,351.412,-86.470,-179.952,16.735,151.553
C07942=1103.885,351.164,-86.436,-179.955,16.732,151.553
C07943=1103.879,350.916,-86.401,-179.958,16.729,151.553
C07944=1103.873,350.668,-86.367,-179.961,16.726,151.553
C07945=1103.868,350.421,-86.333,-179.964,16.723,151.553
C07946=1103.862,350.174,-86.299,-179.967,16.720,151.553
C07947=1103.857,349.926,-86.265,-179.971,16.716,151.553
C07948=1103.851,349.678,-86.231,-179.974,16.714,151.553
C07949=1103.845,349.431,-86.197,-179.976,16.711,151.552
C07950=1103.839,349.184,-86.163,-179.980,16.708,151.552
C07951=1103.834,348.935,-86.129,-179.983,16.705,151.552
C07952=1103.828,348.687,-86.095,-179.986,16.702,151.552
C07953=1103.822,348.440,-86.061,-179.989,16.699,151.552
C07954=1103.817,348.192,-86.027,-179.993,16.696,151.552
C07955=1103.811,347.945,-85.993,-179.995,16.693,151.552
C07956=1103.805,347.698,-85.959,-179.998,16.690,151.552
C07957=1103.800,347.449,-85.925,179.998,16.687,151.552
C07958=1103.794,347.202,-85.891,179.995,16.684,151.552
C07959=1103.789,346.954,-85.858,179.992,16.682,151.552
C07960=1103.783,346.707,-85.824,179.989,16.679,151.552
C07961=1103.777,346.459,-85.791,179.985,16.675,151.552
C07962=1103.771,346.212,-85.757,179.982,16.673,151.552
C07963=1103.766,345.964,-85.723,179.979,16.670,151.552
C07964=1103.760,345.717,-85.689,179.976,16.667,151.552
C07965=1103.754,345.468,-85.655,179.973,16.664,151.552
C07966=1103.749,345.220,-85.621,179.970,16.661,151.551
C07967=1103.743,344.972,-85.587,179.967,16.659,151.551
C07968=1103.737,344.725,-85.553,179.964,16.656,151.551
C07969=1103.731,344.478,-85.521,179.960,16.653,151.551
C07970=1103.725,344.230,-85.487,179.957,16.650,151.551
C07971=1103.720,343.982,-85.453,179.954,16.648,151.551
C07972=1103.711,343.612,-85.403,179.949,16.644,151.551
C07973=1103.703,343.242,-85.354,179.944,16.639,151.551
C07974=1103.694,342.873,-85.303,179.939,16.635,151.551
C07975=1103.686,342.502,-85.253,179.935,16.631,151.551
C07976=1103.681,342.254,-85.219,179.932,16.629,151.551
C07977=1103.675,342.007,-85.185,179.928,16.625,151.551
C07978=1103.668,341.759,-85.153,179.925,16.623,151.551
C07979=1103.663,341.512,-85.119,179.922,16.620,151.551
C07980=1103.657,341.264,-85.086,179.919,16.618,151.551
C07981=1103.652,341.016,-85.053,179.916,16.615,151.551
C07982=1103.646,340.768,-85.019,179.912,16.612,151.551
C07983=1103.640,340.521,-84.985,179.909,16.610,151.551
C07984=1103.635,340.273,-84.952,179.905,16.607,151.551
C07985=1103.629,340.025,-84.919,179.902,16.605,151.551
C07986=1103.624,339.778,-84.886,179.899,16.602,151.551
C07987=1103.618,339.530,-84.853,179.896,16.599,151.551
C07988=1103.612,339.282,-84.819,179.892,16.596,151.551
C07989=1103.607,339.034,-84.786,179.889,16.594,151.551
C07990=1103.601,338.787,-84.752,179.886,16.591,151.551
C07991=1103.595,338.539,-84.719,179.883,16.589,151.552
C07992=1103.589,338.291,-84.686,179.880,16.586,151.552
C07993=1103.584,338.043,-84.653,179.877,16.584,151.552
C07994=1103.578,337.796,-84.619,179.873,16.581,151.552
C07995=1103.572,337.548,-84.587,179.870,16.578,151.552
C07996=1103.566,337.300,-84.553,179.867,16.576,151.552
C07997=1103.561,337.053,-84.520,179.863,16.574,151.552
C07998=1103.556,336.805,-84.487,179.860,16.571,151.552
C07999=1103.550,336.557,-84.455,179.857,16.569,151.552
C08000=1103.544,336.309,-84.422,179.854,16.566,151.552
C08001=1103.539,336.061,-84.388,179.851,16.564,151.552
C08002=1103.532,335.813,-84.355,179.847,16.561,151.552
C08003=1103.527,335.565,-84.322,179.844,16.558,151.552
C08004=1103.521,335.318,-84.289,179.840,16.556,151.552
C08005=1103.516,335.071,-84.256,179.837,16.554,151.553
C08006=1103.510,334.823,-84.223,179.834,16.551,151.553
C08007=1103.504,334.575,-84.191,179.831,16.549,151.553
C08008=1103.498,334.327,-84.158,179.828,16.546,151.553
C08009=1103.493,334.079,-84.124,179.825,16.544,151.553
C08010=1103.487,333.832,-84.092,179.821,16.542,151.553
C08011=1103.482,333.584,-84.059,179.818,16.539,151.553
C08012=1103.476,333.335,-84.026,179.814,16.536,151.553
C08013=1103.470,333.088,-83.993,179.811,16.534,151.553
C08014=1103.465,332.840,-83.960,179.808,16.532,151.553
C08015=1103.459,332.592,-83.928,179.804,16.529,151.553
C08016=1103.454,332.344,-83.895,179.801,16.527,151.553
C08017=1103.447,332.097,-83.862,179.798,16.525,151.554
C08018=1103.442,331.848,-83.830,179.794,16.522,151.554
C08019=1103.436,331.601,-83.797,179.791,16.520,151.554
C08020=1103.430,331.354,-83.764,179.788,16.518,151.554
C08021=1103.425,331.105,-83.732,179.785,16.516,151.554
C08022=1103.419,330.858,-83.699,179.781,16.513,151.554
C08023=1103.413,330.610,-83.666,179.778,16.511,151.554
C08024=1103.404,330.234,-83.617,179.773,16.508,151.555
C08025=1103.395,329.858,-83.567,179.768,16.504,151.555
C08026=1103.387,329.482,-83.518,179.763,16.501,151.555
C08027=1103.378,329.106,-83.469,179.757,16.497,151.555
C08028=1103.372,328.857,-83.436,179.754,16.495,151.555
C08029=1103.366,328.610,-83.403,179.751,16.492,151.555
C08030=1103.361,328.362,-83.372,179.748,16.490,151.556
C08031=1103.354,328.115,-83.339,179.744,16.488,151.556
C08032=1103.349,327.866,-83.306,179.741,16.486,151.556
C08033=1103.343,327.618,-83.274,179.737,16.484,151.556
C08034=1103.338,327.371,-83.242,179.734,16.482,151.556
C08035=1103.332,327.122,-83.209,179.731,16.480,151.557
C08036=1103.326,326.875,-83.177,179.727,16.477,151.557
C08037=1103.321,326.627,-83.145,179.724,16.475,151.557
C08038=1103.315,326.379,-83.113,179.721,16.473,151.557
C08039=1103.309,326.131,-83.080,179.717,16.471,151.557
C08040=1103.304,325.884,-83.048,179.714,16.469,151.557
C08041=1103.298,325.635,-83.016,179.711,16.467,151.558
C08042=1103.291,325.388,-82.983,179.707,16.464,151.558
C08043=1103.287,325.140,-82.951,179.704,16.462,151.558
C08044=1103.281,324.892,-82.919,179.700,16.460,151.558
C08045=1103.275,324.644,-82.887,179.698,16.459,151.558
C08046=1103.269,324.397,-82.854,179.695,16.456,151.558
C08047=1103.263,324.148,-82.822,179.691,16.454,151.559
C08048=1103.258,323.901,-82.790,179.688,16.452,151.559
C08049=1103.252,323.652,-82.758,179.684,16.450,151.559
C08050=1103.246,323.404,-82.726,179.681,16.448,151.559
C08051=1103.241,323.157,-82.694,179.678,16.446,151.559
C08052=1103.235,322.909,-82.662,179.674,16.443,151.559
C08053=1103.229,322.662,-82.630,179.671,16.441,151.560
C08054=1103.223,322.413,-82.598,179.668,16.439,151.560
C08055=1103.218,322.165,-82.565,179.664,16.437,151.560
C08056=1103.213,321.917,-82.534,179.661,16.435,151.560
C08057=1103.207,321.669,-82.502,179.657,16.433,151.560
C08058=1103.201,321.422,-82.470,179.654,16.431,151.561
C08059=1103.195,321.173,-82.438,179.651,16.429,151.561
C08060=1103.190,320.926,-82.406,179.647,16.427,151.561
C08061=1103.184,320.678,-82.374,179.644,16.424,151.561
C08062=1103.179,320.430,-82.343,179.640,16.423,151.562
C08063=1103.173,320.182,-82.310,179.637,16.421,151.562
C08064=1103.168,319.934,-82.278,179.633,16.418,151.562
C08065=1103.162,319.686,-82.246,179.631,16.417,151.562
C08066=1103.157,319.438,-82.215,179.628,16.415,151.562
C08067=1103.151,319.190,-82.183,179.624,16.413,151.563
C08068=1103.145,318.943,-82.151,179.620,16.411,151.563
C08069=1103.139,318.694,-82.119,179.617,16.409,151.563
C08070=1103.134,318.447,-82.087,179.614,16.407,151.563
C08071=1103.128,318.199,-82.055,179.610,16.405,151.563
C08072=1103.123,317.951,-82.024,179.607,16.403,151.564
C08073=1103.117,317.703,-81.993,179.603,16.400,151.564
C08074=1103.111,317.455,-81.961,179.600,16.398,151.564
C08075=1103.106,317.207,-81.929,179.596,16.397,151.564
C08076=1103.098,316.824,-81.880,179.591,16.394,151.565
C08077=1103.089,316.440,-81.831,179.586,16.391,151.565
C08078=1103.080,316.058,-81.782,179.581,16.387,151.565
C08079=1103.072,315.675,-81.733,179.576,16.384,151.566
C08080=1103.066,315.426,-81.702,179.572,16.382,151.566
C08081=1103.061,315.179,-81.670,179.569,16.381,151.566
C08082=1103.054,314.931,-81.639,179.566,16.379,151.566
C08083=1103.049,314.683,-81.607,179.562,16.377,151.567
C08084=1103.043,314.434,-81.576,179.559,16.376,151.567
C08085=1103.038,314.187,-81.544,179.555,16.373,151.567
C08086=1103.031,313.940,-81.513,179.552,16.372,151.568
C08087=1103.026,313.691,-81.482,179.548,16.370,151.568
C08088=1103.020,313.443,-81.450,179.545,16.368,151.568
C08089=1103.014,313.195,-81.419,179.542,16.367,151.568
C08090=1103.009,312.947,-81.388,179.538,16.365,151.569
C08091=1103.003,312.699,-81.356,179.535,16.363,151.569
C08092=1102.997,312.451,-81.325,179.531,16.361,151.569
C08093=1102.991,312.204,-81.294,179.527,16.359,151.570
C08094=1102.985,311.955,-81.263,179.525,16.358,151.570
C08095=1102.980,311.708,-81.231,179.521,16.356,151.570
C08096=1102.974,311.459,-81.200,179.517,16.354,151.571
C08097=1102.968,311.212,-81.169,179.514,16.352,151.571
C08098=1102.963,310.963,-81.138,179.510,16.350,151.571
C08099=1102.957,310.715,-81.106,179.507,16.349,151.571
C08100=1102.951,310.467,-81.076,179.504,16.348,151.572
C08101=1102.946,310.220,-81.044,179.500,16.345,151.572
C08102=1102.939,309.971,-81.013,179.497,16.344,151.572
C08103=1102.934,309.724,-80.982,179.493,16.342,151.573
C08104=1102.928,309.476,-80.951,179.490,16.340,151.573
C08105=1102.922,309.227,-80.920,179.486,16.338,151.573
C08106=1102.917,308.980,-80.888,179.483,16.337,151.573
C08107=1102.911,308.732,-80.858,179.480,16.335,151.574
C08108=1102.906,308.484,-80.826,179.476,16.334,151.574
C08109=1102.899,308.236,-80.796,179.472,16.332,151.574
C08110=1102.894,307.988,-80.765,179.469,16.330,151.575
C08111=1102.888,307.741,-80.734,179.466,16.329,151.575
C08112=1102.882,307.492,-80.702,179.462,16.327,151.575
C08113=1102.877,307.244,-80.672,179.459,16.325,151.576
C08114=1102.871,306.996,-80.641,179.455,16.323,151.576
C08115=1102.865,306.749,-80.610,179.451,16.322,151.576
C08116=1102.860,306.500,-80.579,179.448,16.319,151.577
C08117=1102.854,306.252,-80.548,179.445,16.318,151.577
C08118=1102.849,306.004,-80.517,179.441,16.317,151.577
C08119=1102.843,305.757,-80.486,179.438,16.315,151.578
C08120=1102.838,305.508,-80.455,179.434,16.313,151.578
C08121=1102.832,305.261,-80.425,179.430,16.311,151.578
C08122=1102.826,305.012,-80.394,179.428,16.310,151.579
C08123=1102.820,304.764,-80.363,179.424,16.309,151.579
C08124=1102.814,304.516,-80.333,179.420,16.307,151.579
C08125=1102.809,304.268,-80.302,179.417,16.305,151.580
C08126=1102.803,304.021,-80.271,179.413,16.303,151.580
C08127=1102.798,303.773,-80.240,179.410,16.302,151.580
C08128=1102.789,303.392,-80.193,179.405,16.299,151.581
C08129=1102.780,303.011,-80.146,179.399,16.297,151.581
C08130=1102.772,302.631,-80.099,179.394,16.294,151.582
C08131=1102.763,302.250,-80.052,179.388,16.292,151.582
C08132=1102.758,302.001,-80.022,179.385,16.290,151.583
C08133=1102.752,301.753,-79.991,179.382,16.289,151.583
C08134=1102.747,301.505,-79.961,179.378,16.287,151.583
C08135=1102.741,301.258,-79.930,179.374,16.285,151.584
C08136=1102.736,301.009,-79.899,179.371,16.284,151.584
C08137=1102.730,300.762,-79.869,179.368,16.282,151.584
C08138=1102.724,300.514,-79.839,179.364,16.281,151.585
C08139=1102.719,300.266,-79.808,179.360,16.279,151.585
C08140=1102.713,300.018,-79.777,179.358,16.278,151.585
C08141=1102.707,299.770,-79.747,179.354,16.276,151.586
C08142=1102.702,299.522,-79.716,179.350,16.274,151.586
C08143=1102.697,299.273,-79.686,179.347,16.273,151.586
C08144=1102.691,299.026,-79.656,179.344,16.272,151.587
C08145=1102.685,298.778,-79.626,179.340,16.270,151.587
C08146=1102.680,298.530,-79.595,179.336,16.268,151.588
C08147=1102.674,298.282,-79.564,179.333,16.266,151.588
C08148=1102.669,298.033,-79.535,179.330,16.265,151.588
C08149=1102.663,297.786,-79.504,179.326,16.264,151.589
C08150=1102.657,297.538,-79.474,179.322,16.262,151.589
C08151=1102.652,297.290,-79.443,179.318,16.261,151.589
C08152=1102.646,297.040,-79.413,179.316,16.260,151.590
C08153=1102.640,296.793,-79.383,179.312,16.258,151.590
C08154=1102.634,296.545,-79.352,179.308,16.257,151.591
C08155=1102.629,296.296,-79.323,179.305,16.255,151.591
C08156=1102.623,296.049,-79.292,179.301,16.254,151.591
C08157=1102.617,295.801,-79.262,179.298,16.252,151.592
C08158=1102.612,295.552,-79.232,179.294,16.251,151.592
C08159=1102.606,295.304,-79.202,179.291,16.250,151.593
C08160=1102.600,295.056,-79.172,179.287,16.248,151.593
C08161=1102.595,294.808,-79.142,179.284,16.246,151.593
C08162=1102.589,294.560,-79.112,179.280,16.245,151.594
C08163=1102.583,294.312,-79.082,179.277,16.244,151.594
C08164=1102.577,294.064,-79.052,179.273,16.242,151.594
C08165=1102.572,293.816,-79.022,179.270,16.241,151.595
C08166=1102.566,293.568,-78.992,179.266,16.240,151.595
C08167=1102.561,293.319,-78.962,179.262,16.238,151.596
C08168=1102.555,293.072,-78.932,179.258,16.237,151.596
C08169=1102.550,292.824,-78.903,179.256,16.236,151.597
C08170=1102.544,292.576,-78.872,179.252,16.234,151.597
C08171=1102.538,292.328,-78.843,179.248,16.233,151.597
C08172=1102.533,292.080,-78.812,179.245,16.231,151.598
C08173=1102.527,291.831,-78.783,179.241,16.230,151.598
C08174=1102.522,291.583,-78.753,179.237,16.228,151.599
C08175=1102.516,291.335,-78.723,179.234,16.227,151.599
C08176=1102.510,291.087,-78.693,179.231,16.226,151.599
C08177=1102.504,290.839,-78.664,179.227,16.224,151.600
C08178=1102.498,290.591,-78.634,179.224,16.223,151.600
C08179=1102.493,290.342,-78.604,179.220,16.222,151.601
C08180=1102.485,289.976,-78.560,179.215,16.220,151.601
C08181=1102.476,289.609,-78.516,179.209,16.218,151.602
C08182=1102.468,289.243,-78.472,179.205,16.216,151.602
C08183=1102.460,288.876,-78.428,179.200,16.214,151.603
C08184=1102.454,288.628,-78.398,179.196,16.213,151.604
C08185=1102.448,288.379,-78.369,179.192,16.211,151.604
C08186=1102.442,288.131,-78.340,179.189,16.211,151.605
C08187=1102.436,287.883,-78.309,179.185,16.209,151.605
C08188=1102.431,287.635,-78.280,179.181,16.208,151.605
C08189=1102.425,287.387,-78.251,179.178,16.207,151.606
C08190=1102.419,287.138,-78.221,179.174,16.205,151.606
C08191=1102.414,286.890,-78.192,179.171,16.204,151.607
C08192=1102.409,286.642,-78.162,179.167,16.203,151.607
C08193=1102.402,286.394,-78.133,179.164,16.201,151.608
C08194=1102.397,286.146,-78.103,179.160,16.201,151.608
C08195=1102.391,285.898,-78.073,179.157,16.199,151.609
C08196=1102.385,285.649,-78.044,179.153,16.198,151.609
C08197=1102.380,285.402,-78.015,179.150,16.197,151.609
C08198=1102.374,285.153,-77.985,179.146,16.195,151.610
C08199=1102.368,284.905,-77.956,179.142,16.194,151.610
C08200=1102.363,284.657,-77.927,179.139,16.193,151.611
C08201=1102.357,284.408,-77.897,179.135,16.192,151.611
C08202=1102.352,284.161,-77.868,179.132,16.191,151.612
C08203=1102.346,283.912,-77.839,179.128,16.189,151.612
C08204=1102.341,283.664,-77.809,179.124,16.188,151.613
C08205=1102.334,283.416,-77.780,179.121,16.187,151.613
C08206=1102.329,283.168,-77.751,179.117,16.186,151.613
C08207=1102.323,282.920,-77.722,179.114,16.185,151.614
C08208=1102.318,282.671,-77.692,179.111,16.183,151.614
C08209=1102.312,282.422,-77.663,179.107,16.182,151.615
C08210=1102.307,282.175,-77.634,179.104,16.181,151.615
C08211=1102.301,281.927,-77.605,179.100,16.180,151.616
C08212=1102.296,281.678,-77.575,179.097,16.179,151.616
C08213=1102.289,281.430,-77.546,179.093,16.177,151.617
C08214=1102.285,281.182,-77.517,179.089,16.176,151.617
C08215=1102.278,280.934,-77.488,179.086,16.175,151.617
C08216=1102.273,280.685,-77.459,179.082,16.174,151.618
C08217=1102.267,280.437,-77.430,179.079,16.173,151.619
C08218=1102.261,280.189,-77.401,179.075,16.172,151.619
C08219=1102.256,279.941,-77.371,179.072,16.171,151.619
C08220=1102.250,279.692,-77.343,179.068,16.169,151.620
C08221=1102.245,279.445,-77.314,179.064,16.168,151.620
C08222=1102.239,279.196,-77.285,179.061,16.167,151.621
C08223=1102.233,278.948,-77.255,179.057,16.166,151.621
C08224=1102.227,278.699,-77.227,179.054,16.165,151.622
C08225=1102.222,278.451,-77.198,179.050,16.164,151.622
C08226=1102.216,278.203,-77.169,179.047,16.163,151.623
C08227=1102.210,277.955,-77.140,179.043,16.161,151.623
C08228=1102.205,277.707,-77.111,179.039,16.160,151.624
C08229=1102.199,277.459,-77.082,179.036,16.159,151.624
C08230=1102.194,277.210,-77.053,179.032,16.158,151.625
C08231=1102.188,276.962,-77.024,179.029,16.157,151.625
C08232=1102.179,276.605,-76.983,179.024,16.156,151.626
C08233=1102.172,276.248,-76.941,179.018,16.153,151.627
C08234=1102.163,275.890,-76.900,179.013,16.152,151.627
C08235=1102.156,275.532,-76.859,179.008,16.151,151.628
C08236=1102.149,275.284,-76.830,179.005,16.150,151.629
C08237=1102.144,275.036,-76.802,179.001,16.149,151.629
C08238=1102.138,274.788,-76.772,178.997,16.148,151.630
C08239=1102.133,274.539,-76.744,178.993,16.147,151.630
C08240=1102.127,274.291,-76.715,178.990,16.146,151.631
C08241=1102.121,274.043,-76.687,178.987,16.144,151.631
C08242=1102.116,273.795,-76.658,178.983,16.143,151.632
C08243=1102.110,273.546,-76.629,178.979,16.142,151.632
C08244=1102.104,273.299,-76.601,178.975,16.141,151.633
C08245=1102.099,273.050,-76.572,178.972,16.141,151.633
C08246=1102.093,272.801,-76.544,178.968,16.139,151.634
C08247=1102.088,272.553,-76.515,178.965,16.139,151.634
C08248=1102.082,272.305,-76.486,178.961,16.137,151.635
C08249=1102.076,272.057,-76.458,178.958,16.136,151.635
C08250=1102.070,271.808,-76.429,178.954,16.135,151.636
C08251=1102.065,271.560,-76.401,178.951,16.134,151.636
C08252=1102.059,271.312,-76.373,178.947,16.133,151.637
C08253=1102.054,271.063,-76.344,178.944,16.132,151.637
C08254=1102.048,270.815,-76.315,178.940,16.131,151.638
C08255=1102.042,270.566,-76.287,178.937,16.131,151.638
C08256=1102.037,270.318,-76.259,178.933,16.129,151.639
C08257=1102.031,270.070,-76.231,178.929,16.129,151.639
C08258=1102.025,269.822,-76.202,178.925,16.127,151.640
C08259=1102.019,269.573,-76.174,178.922,16.127,151.640
C08260=1102.014,269.325,-76.146,178.918,16.125,151.641
C08261=1102.008,269.077,-76.118,178.915,16.125,151.641
C08262=1102.003,268.829,-76.090,178.911,16.124,151.642
C08263=1101.996,268.580,-76.061,178.908,16.123,151.642
C08264=1101.991,268.332,-76.033,178.904,16.122,151.643
C08265=1101.985,268.084,-76.004,178.901,16.121,151.643
C08266=1101.980,267.836,-75.976,178.897,16.120,151.644
C08267=1101.974,267.587,-75.947,178.893,16.119,151.644
C08268=1101.969,267.339,-75.919,178.889,16.118,151.645
C08269=1101.962,267.090,-75.892,178.886,16.117,151.646
C08270=1101.957,266.842,-75.864,178.882,16.116,151.646
C08271=1101.951,266.593,-75.835,178.879,16.115,151.647
C08272=1101.946,266.345,-75.808,178.875,16.114,151.647
C08273=1101.940,266.096,-75.779,178.872,16.113,151.648
C08274=1101.935,265.848,-75.751,178.868,16.112,151.648
C08275=1101.929,265.600,-75.723,178.865,16.112,151.649
C08276=1101.923,265.352,-75.695,178.861,16.110,151.649
C08277=1101.918,265.104,-75.667,178.857,16.110,151.650
C08278=1101.912,264.855,-75.639,178.853,16.108,151.650
C08279=1101.907,264.607,-75.611,178.850,16.108,151.651
C08280=1101.901,264.358,-75.582,178.846,16.107,151.651
C08281=1101.895,264.110,-75.554,178.843,16.106,151.652
C08282=1101.889,263.861,-75.526,178.840,16.105,151.652
C08283=1101.883,263.613,-75.499,178.836,16.104,151.653
C08284=1101.876,263.258,-75.459,178.830,16.103,151.654
C08285=1101.867,262.904,-75.419,178.825,16.101,151.655
C08286=1101.859,262.549,-75.379,178.820,16.100,151.655
C08287=1101.850,262.195,-75.340,178.815,16.099,151.656
C08288=1101.845,261.946,-75.312,178.811,16.099,151.657
C08289=1101.840,261.698,-75.284,178.807,16.098,151.657
C08290=1101.833,261.450,-75.257,178.804,16.097,151.658
C08291=1101.828,261.202,-75.229,178.801,16.096,151.658
C08292=1101.822,260.952,-75.201,178.797,16.095,151.659
C08293=1101.817,260.704,-75.173,178.794,16.095,151.660
C08294=1101.811,260.457,-75.146,178.790,16.094,151.660
C08295=1101.805,260.208,-75.117,178.786,16.093,151.661
C08296=1101.800,259.959,-75.090,178.782,16.092,151.661
C08297=1101.793,259.711,-75.062,178.779,16.091,151.662
C08298=1101.788,259.463,-75.034,178.776,16.091,151.662
C08299=1101.783,259.214,-75.007,178.772,16.090,151.663
C08300=1101.776,258.965,-74.979,178.768,16.089,151.664
C08301=1101.770,258.717,-74.952,178.764,16.088,151.664
C08302=1101.765,258.469,-74.925,178.761,16.087,151.665
C08303=1101.759,258.220,-74.897,178.757,16.086,151.665
C08304=1101.754,257.972,-74.869,178.754,16.086,151.666
C08305=1101.748,257.724,-74.842,178.750,16.085,151.666
C08306=1101.742,257.475,-74.814,178.746,16.084,151.667
C08307=1101.737,257.226,-74.786,178.743,16.083,151.667
C08308=1101.731,256.978,-74.760,178.739,16.082,151.668
C08309=1101.725,256.729,-74.731,178.736,16.082,151.669
C08310=1101.719,256.481,-74.705,178.732,16.081,151.669
C08311=1101.714,256.233,-74.677,178.729,16.080,151.670
C08312=1101.708,255.985,-74.650,178.725,16.080,151.670
C08313=1101.702,255.736,-74.622,178.721,16.078,151.671
C08314=1101.697,255.487,-74.595,178.718,16.078,151.671
C08315=1101.691,255.239,-74.567,178.714,16.077,151.672
C08316=1101.686,254.991,-74.540,178.711,16.076,151.673
C08317=1101.679,254.742,-74.512,178.707,16.076,151.673
C08318=1101.674,254.494,-74.485,178.703,16.075,151.674
C08319=1101.668,254.245,-74.458,178.700,16.074,151.674
C08320=1101.663,253.997,-74.430,178.696,16.073,151.675
C08321=1101.657,253.748,-74.403,178.693,16.072,151.675
C08322=1101.652,253.500,-74.376,178.688,16.071,151.676
C08323=1101.646,253.252,-74.349,178.685,16.071,151.677
C08324=1101.641,253.003,-74.322,178.682,16.070,151.677
C08325=1101.635,252.755,-74.295,178.678,16.069,151.678
C08326=1101.629,252.506,-74.267,178.674,16.069,151.678
C08327=1101.623,252.258,-74.240,178.670,16.067,151.679
C08328=1101.618,252.009,-74.213,178.667,16.067,151.679
C08329=1101.612,251.761,-74.186,178.664,16.066,151.680
C08330=1101.607,251.513,-74.158,178.660,16.065,151.681
C08331=1101.601,251.264,-74.131,178.656,16.065,151.681
C08332=1101.596,251.015,-74.104,178.653,16.064,151.682
C08333=1101.590,250.766,-74.077,178.649,16.063,151.682
C08334=1101.585,250.518,-74.050,178.646,16.062,151.683
C08335=1101.579,250.269,-74.023,178.642,16.061,151.683
C08336=1101.571,249.913,-73.984,178.637,16.060,151.684
C08337=1101.563,249.555,-73.945,178.632,16.060,151.685
C08338=1101.555,249.198,-73.906,178.627,16.058,151.686
C08339=1101.547,248.840,-73.868,178.622,16.057,151.687
C08340=1101.541,248.592,-73.840,178.618,16.057,151.687
C08341=1101.536,248.343,-73.813,178.614,16.055,151.688
C08342=1101.530,248.095,-73.787,178.611,16.055,151.689
C08343=1101.525,247.846,-73.759,178.607,16.054,151.689
C08344=1101.519,247.598,-73.733,178.604,16.053,151.690
C08345=1101.514,247.349,-73.705,178.600,16.053,151.690
C08346=1101.508,247.101,-73.679,178.596,16.052,151.691
C08347=1101.502,246.852,-73.652,178.593,16.051,151.691
C08348=1101.497,246.604,-73.625,178.590,16.051,151.692
C08349=1101.492,246.355,-73.598,178.585,16.050,151.693
C08350=1101.486,246.107,-73.572,178.582,16.049,151.693
C08351=1101.479,245.858,-73.545,178.579,16.049,151.694
C08352=1101.474,245.609,-73.519,178.575,16.048,151.694
C08353=1101.468,245.361,-73.492,178.571,16.047,151.695
C08354=1101.463,245.112,-73.465,178.567,16.046,151.695
C08355=1101.457,244.864,-73.438,178.564,16.046,151.696
C08356=1101.452,244.615,-73.411,178.561,16.045,151.697
C08357=1101.446,244.367,-73.385,178.557,16.044,151.697
C08358=1101.440,244.119,-73.358,178.553,16.044,151.698
C08359=1101.435,243.870,-73.331,178.550,16.043,151.698
C08360=1101.430,243.621,-73.305,178.546,16.042,151.699
C08361=1101.424,243.373,-73.278,178.542,16.042,151.700
C08362=1101.418,243.124,-73.252,178.539,16.041,151.700
C08363=1101.412,242.876,-73.225,178.535,16.041,151.701
C08364=1101.407,242.627,-73.199,178.532,16.040,151.702
C08365=1101.401,242.379,-73.172,178.528,16.039,151.702
C08366=1101.395,242.130,-73.146,178.524,16.039,151.703
C08367=1101.389,241.882,-73.119,178.521,16.038,151.703
C08368=1101.384,241.633,-73.093,178.517,16.038,151.704
C08369=1101.378,241.384,-73.067,178.513,16.037,151.705
C08370=1101.372,241.136,-73.040,178.510,16.036,151.705
C08371=1101.367,240.887,-73.013,178.507,16.036,151.706
C08372=1101.362,240.638,-72.987,178.503,16.035,151.706
C08373=1101.356,240.390,-72.960,178.499,16.034,151.707
C08374=1101.350,240.142,-72.933,178.496,16.034,151.708
C08375=1101.345,239.893,-72.908,178.492,16.034,151.708
C08376=1101.338,239.645,-72.881,178.488,16.032,151.709
C08377=1101.333,239.396,-72.856,178.485,16.032,151.709
C08378=1101.327,239.147,-72.829,178.482,16.032,151.710
C08379=1101.321,238.899,-72.802,178.478,16.031,151.711
C08380=1101.316,238.650,-72.776,178.474,16.030,151.711
C08381=1101.310,238.402,-72.750,178.471,16.030,151.712
C08382=1101.305,238.153,-72.724,178.467,16.029,151.713
C08383=1101.299,237.904,-72.697,178.463,16.028,151.713
C08384=1101.294,237.656,-72.672,178.460,16.028,151.714
C08385=1101.288,237.408,-72.645,178.457,16.028,151.714
C08386=1101.283,237.159,-72.619,178.453,16.026,151.715
C08387=1101.277,236.910,-72.592,178.449,16.026,151.716
C08388=1101.268,236.546,-72.555,178.444,16.025,151.716
C08389=1101.260,236.182,-72.516,178.438,16.024,151.717
C08390=1101.252,235.817,-72.477,178.433,16.023,151.718
C08391=1101.244,235.453,-72.440,178.428,16.023,151.719
C08392=1101.238,235.205,-72.413,178.424,16.022,151.720
C08393=1101.232,234.956,-72.387,178.421,16.022,151.720
C08394=1101.227,234.707,-72.361,178.418,16.021,151.721
C08395=1101.222,234.459,-72.335,178.413,16.020,151.722
C08396=1101.216,234.210,-72.309,178.410,16.020,151.722
C08397=1101.210,233.962,-72.284,178.406,16.020,151.723
C08398=1101.204,233.713,-72.257,178.403,16.019,151.723
C08399=1101.199,233.464,-72.231,178.399,16.018,151.724
C08400=1101.193,233.215,-72.205,178.396,16.018,151.725
C08401=1101.187,232.968,-72.180,178.392,16.017,151.725
C08402=1101.182,232.719,-72.154,178.389,16.017,151.726
C08403=1101.176,232.470,-72.128,178.385,16.016,151.727
C08404=1101.171,232.221,-72.102,178.381,16.015,151.727
C08405=1101.164,231.973,-72.076,178.378,16.015,151.728
C08406=1101.160,231.725,-72.050,178.375,16.015,151.728
C08407=1101.154,231.476,-72.024,178.371,16.014,151.729
C08408=1101.149,231.227,-71.998,178.367,16.013,151.730
C08409=1101.142,230.978,-71.973,178.364,16.013,151.730
C08410=1101.137,230.729,-71.947,178.360,16.012,151.731
C08411=1101.132,230.481,-71.921,178.356,16.011,151.732
C08412=1101.126,230.233,-71.895,178.353,16.011,151.732
C08413=1101.120,229.984,-71.870,178.350,16.011,151.733
C08414=1101.114,229.735,-71.844,178.345,16.010,151.733
C08415=1101.108,229.486,-71.818,178.342,16.010,151.734
C08416=1101.104,229.238,-71.793,178.339,16.009,151.735
C08417=1101.097,228.989,-71.767,178.335,16.009,151.735
C08418=1101.092,228.740,-71.741,178.332,16.009,151.736
C08419=1101.086,228.492,-71.716,178.327,16.008,151.737
C08420=1101.081,228.243,-71.691,178.324,16.007,151.737
C08421=1101.075,227.995,-71.665,178.321,16.007,151.738
C08422=1101.069,227.746,-71.639,178.317,16.006,151.738
C08423=1101.063,227.497,-71.614,178.313,16.006,151.739
C08424=1101.058,227.249,-71.588,178.310,16.006,151.740
C08425=1101.052,227.000,-71.563,178.306,16.005,151.740
C08426=1101.046,226.751,-71.537,178.303,16.005,151.741
C08427=1101.040,226.502,-71.512,178.299,16.004,151.742
C08428=1101.035,226.254,-71.486,178.295,16.003,151.742
C08429=1101.029,226.005,-71.461,178.292,16.003,151.743
C08430=1101.024,225.756,-71.435,178.289,16.003,151.744
C08431=1101.018,225.508,-71.410,178.285,16.002,151.744
C08432=1101.013,225.259,-71.384,178.281,16.001,151.745
C08433=1101.006,225.011,-71.359,178.278,16.001,151.745
C08434=1101.002,224.762,-71.333,178.274,16.001,151.746
C08435=1100.995,224.514,-71.308,178.271,16.000,151.747
C08436=1100.990,224.264,-71.283,178.267,15.999,151.747
C08437=1100.985,224.016,-71.258,178.263,15.999,151.748
C08438=1100.979,223.767,-71.232,178.260,15.999,151.749
C08439=1100.973,223.519,-71.206,178.256,15.999,151.749
C08440=1100.965,223.146,-71.168,178.251,15.998,151.750
C08441=1100.957,222.773,-71.131,178.246,15.997,151.751
C08442=1100.948,222.401,-71.093,178.240,15.996,151.752
C08443=1100.940,222.028,-71.055,178.235,15.996,151.753
C08444=1100.934,221.780,-71.030,178.231,15.995,151.754
C08445=1100.928,221.530,-71.005,178.228,15.995,151.754
C08446=1100.923,221.282,-70.980,178.224,15.994,151.755
C08447=1100.917,221.033,-70.954,178.221,15.994,151.756
C08448=1100.911,220.785,-70.929,178.217,15.994,151.756
C08449=1100.906,220.536,-70.904,178.213,15.993,151.757
C08450=1100.900,220.287,-70.879,178.210,15.992,151.758
C08451=1100.894,220.038,-70.855,178.206,15.992,151.758
C08452=1100.888,219.790,-70.829,178.203,15.992,151.759
C08453=1100.883,219.541,-70.804,178.200,15.992,151.760
C08454=1100.877,219.292,-70.779,178.196,15.990,151.760
C08455=1100.871,219.044,-70.754,178.192,15.990,151.761
C08456=1100.866,218.795,-70.729,178.189,15.990,151.762
C08457=1100.860,218.546,-70.704,178.185,15.990,151.762
C08458=1100.855,218.298,-70.679,178.182,15.989,151.763
C08459=1100.849,218.049,-70.654,178.179,15.989,151.763
C08460=1100.843,217.801,-70.629,178.174,15.988,151.764
C08461=1100.837,217.551,-70.604,178.171,15.988,151.765
C08462=1100.833,217.303,-70.579,178.167,15.987,151.765
C08463=1100.827,217.054,-70.554,178.164,15.987,151.766
C08464=1100.821,216.806,-70.529,178.161,15.987,151.767
C08465=1100.815,216.557,-70.505,178.157,15.987,151.767
C08466=1100.810,216.308,-70.480,178.153,15.986,151.768
C08467=1100.804,216.059,-70.455,178.150,15.985,151.769
C08468=1100.799,215.810,-70.430,178.146,15.985,151.769
C08469=1100.793,215.562,-70.405,178.143,15.985,151.770
C08470=1100.788,215.313,-70.381,178.139,15.985,151.771
C08471=1100.781,215.065,-70.355,178.136,15.984,151.771
C08472=1100.776,214.816,-70.331,178.132,15.983,151.772
C08473=1100.770,214.567,-70.306,178.128,15.983,151.773
C08474=1100.765,214.319,-70.281,178.125,15.983,151.773
C08475=1100.759,214.069,-70.257,178.121,15.982,151.774
C08476=1100.754,213.821,-70.232,178.118,15.982,151.774
C08477=1100.748,213.572,-70.207,178.115,15.982,151.775
C08478=1100.743,213.323,-70.182,178.110,15.981,151.776
C08479=1100.737,213.074,-70.158,178.107,15.980,151.776
C08480=1100.731,212.825,-70.133,178.104,15.980,151.777
C08481=1100.726,212.577,-70.108,178.100,15.980,151.778
C08482=1100.720,212.328,-70.084,178.097,15.980,151.778
C08483=1100.715,212.080,-70.060,178.093,15.980,151.779
C08484=1100.709,211.830,-70.035,178.090,15.979,151.780
C08485=1100.703,211.582,-70.010,178.086,15.978,151.780
C08486=1100.698,211.334,-69.986,178.082,15.978,151.781
C08487=1100.692,211.084,-69.961,178.079,15.978,151.782
C08488=1100.687,210.836,-69.937,178.075,15.978,151.782
C08489=1100.680,210.587,-69.913,178.072,15.977,151.783
C08490=1100.674,210.339,-69.888,178.069,15.977,151.784
C08491=1100.668,210.090,-69.863,178.065,15.977,151.784
C08492=1100.661,209.721,-69.827,178.060,15.976,151.785
C08493=1100.652,209.352,-69.791,178.054,15.975,151.786
C08494=1100.644,208.983,-69.754,178.049,15.975,151.787
C08495=1100.636,208.614,-69.718,178.044,15.974,151.788
C08496=1100.613,207.607,-69.621,178.006,15.964,151.794
C08497=1100.607,207.359,-69.597,178.002,15.965,151.795
C08498=1100.602,207.110,-69.573,177.998,15.965,151.796
C08499=1100.596,206.861,-69.548,177.995,15.965,151.796
C08500=1100.590,206.613,-69.524,177.991,15.966,151.797
C08501=1100.584,206.364,-69.500,177.987,15.966,151.798
C08502=1100.579,206.116,-69.476,177.984,15.967,151.799
C08503=1100.572,205.867,-69.452,177.980,15.968,151.800
C08504=1100.567,205.618,-69.428,177.976,15.968,151.801
C08505=1100.562,205.369,-69.404,177.972,15.968,151.802
C08506=1100.556,205.120,-69.379,177.968,15.969,151.803
C08507=1100.550,204.871,-69.356,177.964,15.969,151.804
C08508=1100.545,204.623,-69.332,177.961,15.970,151.805
C08509=1100.540,204.374,-69.307,177.957,15.970,151.805
C08510=1100.534,204.125,-69.284,177.954,15.971,151.806
C08511=1100.528,203.876,-69.260,177.950,15.971,151.807
C08512=1100.522,203.628,-69.236,177.946,15.972,151.808
C08513=1100.517,203.379,-69.212,177.942,15.972,151.809
C08514=1100.512,203.130,-69.188,177.939,15.973,151.810
C08515=1100.505,202.881,-69.164,177.935,15.973,151.811
C08516=1100.500,202.632,-69.140,177.931,15.974,151.812
C08517=1100.494,202.384,-69.116,177.927,15.974,151.812
C08518=1100.489,202.135,-69.093,177.924,15.974,151.813
C08519=1100.482,201.886,-69.069,177.920,15.975,151.814
C08520=1100.477,201.637,-69.045,177.916,15.976,151.815
C08521=1100.471,201.388,-69.022,177.912,15.976,151.816
C08522=1100.466,201.140,-68.997,177.909,15.977,151.817
C08523=1100.459,200.891,-68.973,177.905,15.977,151.818
C08524=1100.454,200.642,-68.950,177.902,15.978,151.819
C08525=1100.448,200.393,-68.926,177.898,15.978,151.820
C08526=1100.442,200.144,-68.903,177.894,15.979,151.820
C08527=1100.437,199.896,-68.879,177.890,15.979,151.821
C08528=1100.430,199.647,-68.855,177.886,15.979,151.822
C08529=1100.425,199.398,-68.831,177.882,15.980,151.823
C08530=1100.419,199.149,-68.808,177.879,15.981,151.824
C08531=1100.414,198.900,-68.784,177.875,15.981,151.825
C08532=1100.408,198.652,-68.760,177.872,15.982,151.826
C08533=1100.402,198.402,-68.737,177.868,15.982,151.827
C08534=1100.397,198.154,-68.713,177.864,15.982,151.827
C08535=1100.391,197.905,-68.690,177.861,15.983,151.828
C08536=1100.385,197.657,-68.666,177.857,15.984,151.829
C08537=1100.380,197.407,-68.643,177.853,15.984,151.830
C08538=1100.374,197.159,-68.619,177.849,15.984,151.831
C08539=1100.369,196.910,-68.596,177.845,15.985,151.832
C08540=1100.362,196.661,-68.572,177.842,15.986,151.833
C08541=1100.357,196.412,-68.549,177.839,15.986,151.834
C08542=1100.351,196.163,-68.524,177.835,15.986,151.834
C08543=1100.346,195.914,-68.501,177.831,15.986,151.835
C08544=1100.340,195.666,-68.478,177.827,15.987,151.836
C08545=1100.334,195.417,-68.454,177.824,15.988,151.837
C08546=1100.329,195.168,-68.431,177.820,15.988,151.838
C08547=1100.323,194.919,-68.408,177.817,15.988,151.839
C08548=1100.318,194.671,-68.384,177.813,15.989,151.840
C08549=1100.312,194.422,-68.361,177.809,15.989,151.840
C08550=1100.306,194.172,-68.338,177.806,15.990,151.841
C08551=1100.300,193.924,-68.314,177.802,15.990,151.842
C08552=1100.295,193.675,-68.291,177.798,15.990,151.843
C08553=1100.289,193.426,-68.268,177.794,15.991,151.844
C08554=1100.283,193.177,-68.244,177.791,15.992,151.845
C08555=1100.278,192.928,-68.220,177.788,15.992,151.846
C08556=1100.272,192.679,-68.197,177.784,15.993,151.846
C08557=1100.266,192.407,-68.172,177.780,15.993,151.847
C08558=1100.260,192.133,-68.146,177.776,15.993,151.848
C08559=1100.253,191.861,-68.121,177.772,15.994,151.849
C08560=1100.248,191.588,-68.096,177.768,15.995,151.850
C08561=1100.242,191.339,-68.072,177.764,15.994,151.851
C08562=1100.237,191.090,-68.049,177.761,15.995,151.852
C08563=1100.231,190.841,-68.026,177.757,15.995,151.853
C08564=1100.225,190.592,-68.003,177.754,15.996,151.853
C08565=1100.219,190.343,-67.980,177.750,15.996,151.854
C08566=1100.214,190.094,-67.956,177.746,15.997,151.855
C08567=1100.209,189.845,-67.933,177.742,15.997,151.856
C08568=1100.203,189.597,-67.910,177.739,15.997,151.857
C08569=1100.197,189.348,-67.887,177.736,15.998,151.858
C08570=1100.191,189.099,-67.864,177.732,15.998,151.858
C08571=1100.186,188.850,-67.840,177.728,15.999,151.859
C08572=1100.180,188.601,-67.817,177.725,15.999,151.860
C08573=1100.175,188.352,-67.794,177.721,16.000,151.861
C08574=1100.169,188.103,-67.772,177.718,15.999,151.862
C08575=1100.163,187.854,-67.749,177.714,16.000,151.862
C08576=1100.158,187.605,-67.725,177.710,16.000,151.863
C08577=1100.153,187.357,-67.702,177.707,16.000,151.864
C08578=1100.147,187.108,-67.680,177.704,16.001,151.865
C08579=1100.142,186.859,-67.657,177.700,16.002,151.866
C08580=1100.136,186.610,-67.634,177.696,16.002,151.867
C08581=1100.130,186.361,-67.611,177.692,16.002,151.867
C08582=1100.125,186.112,-67.588,177.689,16.002,151.868
C08583=1100.120,185.863,-67.564,177.686,16.003,151.869
C08584=1100.114,185.614,-67.541,177.682,16.003,151.870
C08585=1100.109,185.366,-67.519,177.678,16.003,151.871
C08586=1100.103,185.117,-67.496,177.674,16.004,151.872
C08587=1100.098,184.868,-67.473,177.671,16.005,151.872
C08588=1100.092,184.619,-67.451,177.668,16.005,151.873
C08589=1100.085,184.370,-67.428,177.664,16.005,151.874
C08590=1100.080,184.121,-67.405,177.660,16.005,151.875
C08591=1100.074,183.873,-67.382,177.657,16.006,151.876
C08592=1100.068,183.624,-67.359,177.654,16.006,151.876
C08593=1100.062,183.375,-67.336,177.650,16.007,151.877
C08594=1100.057,183.125,-67.314,177.646,16.007,151.878
C08595=1100.050,182.877,-67.292,177.643,16.008,151.879
C08596=1100.045,182.628,-67.269,177.639,16.008,151.880
C08597=1100.039,182.379,-67.246,177.635,16.008,151.881
C08598=1100.033,182.130,-67.223,177.632,16.008,151.881
C08599=1100.028,181.880,-67.201,177.629,16.009,151.882
C08600=1100.022,181.633,-67.179,177.625,16.010,151.883
C08601=1100.016,181.384,-67.156,177.621,16.010,151.884
C08602=1100.011,181.135,-67.133,177.617,16.010,151.885
C08603=1100.005,180.885,-67.111,177.614,16.011,151.886
C08604=1099.999,180.636,-67.088,177.611,16.011,151.886
C08605=1099.993,180.388,-67.065,177.607,16.011,151.887
C08606=1099.987,180.139,-67.042,177.603,16.011,151.888
C08607=1099.982,179.889,-67.020,177.600,16.012,151.889
C08608=1099.977,179.641,-66.998,177.596,16.013,151.890
C08609=1099.970,179.393,-66.975,177.593,16.013,151.890
C08610=1099.965,179.143,-66.953,177.589,16.013,151.891
C08611=1099.959,178.894,-66.930,177.586,16.014,151.892
C08612=1099.953,178.645,-66.907,177.582,16.014,151.893
C08613=1099.947,178.396,-66.885,177.579,16.014,151.894
C08614=1099.942,178.148,-66.863,177.576,16.015,151.895
C08615=1099.937,177.898,-66.841,177.572,16.015,151.895
C08616=1099.931,177.649,-66.818,177.568,16.016,151.896
C08617=1099.924,177.401,-66.795,177.565,16.015,151.897
C08618=1099.919,177.151,-66.773,177.562,16.017,151.898
C08619=1099.914,176.903,-66.751,177.558,16.016,151.898
C08620=1099.908,176.654,-66.729,177.554,16.017,151.899
C08621=1099.902,176.381,-66.704,177.551,16.017,151.900
C08622=1099.895,176.107,-66.679,177.547,16.018,151.901
C08623=1099.889,175.834,-66.655,177.543,16.018,151.902
C08624=1099.883,175.560,-66.630,177.539,16.018,151.903
C08625=1099.877,175.311,-66.609,177.535,16.018,151.904
C08626=1099.871,175.062,-66.586,177.533,16.019,151.904
C08627=1099.866,174.813,-66.563,177.529,16.019,151.905
C08628=1099.860,174.565,-66.541,177.525,16.019,151.906
C08629=1099.855,174.315,-66.519,177.522,16.019,151.907
C08630=1099.849,174.066,-66.498,177.519,16.020,151.908
C08631=1099.843,173.817,-66.475,177.515,16.020,151.908
C08632=1099.838,173.569,-66.453,177.511,16.021,151.909
C08633=1099.832,173.320,-66.430,177.508,16.021,151.910
C08634=1099.826,173.070,-66.408,177.505,16.021,151.911
C08635=1099.821,172.822,-66.386,177.501,16.022,151.911
C08636=1099.815,172.573,-66.364,177.497,16.022,151.912
C08637=1099.809,172.324,-66.342,177.495,16.022,151.913
C08638=1099.804,172.075,-66.320,177.491,16.023,151.914
C08639=1099.798,171.826,-66.298,177.487,16.023,151.915
C08640=1099.793,171.577,-66.275,177.484,16.023,151.915
C08641=1099.787,171.328,-66.254,177.481,16.023,151.916
C08642=1099.781,171.079,-66.231,177.477,16.024,151.917
C08643=1099.775,170.830,-66.209,177.474,16.024,151.918
C08644=1099.770,170.581,-66.188,177.470,16.024,151.918
C08645=1099.764,170.332,-66.166,177.467,16.024,151.919
C08646=1099.759,170.084,-66.143,177.463,16.025,151.920
C08647=1099.754,169.834,-66.121,177.460,16.025,151.921
C08648=1099.748,169.585,-66.099,177.457,16.025,151.921
C08649=1099.743,169.336,-66.078,177.453,16.025,151.922
C08650=1099.737,169.087,-66.056,177.450,16.026,151.923
C08651=1099.731,168.839,-66.033,177.446,16.026,151.924
C08652=1099.725,168.590,-66.012,177.443,16.026,151.924
C08653=1099.720,168.340,-65.990,177.440,16.026,151.925
C08654=1099.714,168.092,-65.968,177.436,16.026,151.926
C08655=1099.709,167.842,-65.946,177.433,16.027,151.927
C08656=1099.703,167.594,-65.925,177.430,16.027,151.927
C08657=1099.698,167.345,-65.902,177.426,16.027,151.928
C08658=1099.692,167.096,-65.881,177.422,16.027,151.929
C08659=1099.687,166.847,-65.858,177.420,16.028,151.930
C08660=1099.680,166.597,-65.837,177.416,16.028,151.930
C08661=1099.676,166.349,-65.815,177.413,16.028,151.931
C08662=1099.669,166.099,-65.793,177.409,16.028,151.932
C08663=1099.665,165.851,-65.771,177.406,16.028,151.933
C08664=1099.658,165.601,-65.750,177.402,16.029,151.933
C08665=1099.654,165.353,-65.728,177.399,16.029,151.934
C08666=1099.647,165.103,-65.706,177.396,16.029,151.935
C08667=1099.643,164.855,-65.684,177.392,16.029,151.936
C08668=1099.636,164.605,-65.663,177.389,16.029,151.936
C08669=1099.632,164.357,-65.641,177.385,16.029,151.937
C08670=1099.625,164.107,-65.619,177.383,16.030,151.938
C08671=1099.621,163.859,-65.597,177.379,16.030,151.938
C08672=1099.614,163.609,-65.576,177.375,16.030,151.939
C08673=1099.609,163.361,-65.554,177.373,16.030,151.940
C08674=1099.604,163.112,-65.533,177.369,16.030,151.941
C08675=1099.598,162.863,-65.511,177.366,16.030,151.941
C08676=1099.593,162.614,-65.489,177.362,16.030,151.942
C08677=1099.587,162.364,-65.468,177.359,16.031,151.943
C08678=1099.582,162.116,-65.447,177.356,16.031,151.944
C08679=1099.576,161.866,-65.425,177.352,16.031,151.944
C08680=1099.571,161.618,-65.403,177.349,16.031,151.945
C08681=1099.565,161.368,-65.382,177.346,16.031,151.946
C08682=1099.560,161.120,-65.360,177.342,16.031,151.946
C08683=1099.554,160.870,-65.338,177.339,16.032,151.947
C08684=1099.548,160.622,-65.317,177.336,16.032,151.948
C08685=1099.542,160.348,-65.293,177.332,16.032,151.949
C08686=1099.536,160.073,-65.270,177.329,16.032,151.950
C08687=1099.530,159.800,-65.247,177.325,16.032,151.950
C08688=1099.523,159.526,-65.224,177.321,16.033,151.951
C08689=1099.518,159.278,-65.202,177.318,16.033,151.952
C08690=1099.512,159.028,-65.180,177.315,16.033,151.953
C08691=1099.506,158.780,-65.159,177.311,16.033,151.953
C08692=1099.501,158.530,-65.138,177.308,16.033,151.954
C08693=1099.495,158.281,-65.117,177.305,16.033,151.955
C08694=1099.489,158.032,-65.095,177.302,16.033,151.955
C08695=1099.483,157.784,-65.074,177.298,16.033,151.956
C08696=1099.479,157.534,-65.053,177.295,16.034,151.957
C08697=1099.473,157.285,-65.031,177.292,16.034,151.958
C08698=1099.467,157.037,-65.010,177.288,16.034,151.958
C08699=1099.461,156.787,-64.989,177.285,16.034,151.959
C08700=1099.456,156.538,-64.968,177.282,16.035,151.960
C08701=1099.449,156.289,-64.946,177.278,16.035,151.960
C08702=1099.444,156.040,-64.925,177.275,16.035,151.961
C08703=1099.439,155.791,-64.904,177.272,16.035,151.962
C08704=1099.433,155.542,-64.882,177.269,16.035,151.962
C08705=1099.427,155.293,-64.862,177.265,16.035,151.963
C08706=1099.422,155.045,-64.841,177.262,16.035,151.964
C08707=1099.417,154.794,-64.819,177.259,16.035,151.965
C08708=1099.411,154.546,-64.798,177.255,16.035,151.965
C08709=1099.405,154.297,-64.776,177.252,16.036,151.966
C08710=1099.400,154.048,-64.756,177.249,16.036,151.967
C08711=1099.394,153.799,-64.734,177.245,16.036,151.968
C08712=1099.388,153.549,-64.713,177.243,16.036,151.968
C08713=1099.383,153.301,-64.692,177.239,16.036,151.969
C08714=1099.377,153.052,-64.672,177.236,16.036,151.970
C08715=1099.371,152.802,-64.650,177.233,16.037,151.970
C08716=1099.365,152.554,-64.630,177.229,16.037,151.971
C08717=1099.360,152.305,-64.609,177.226,16.036,151.972
C08718=1099.354,152.055,-64.588,177.223,16.037,151.972
C08719=1099.348,151.807,-64.567,177.220,16.037,151.973
C08720=1099.343,151.558,-64.546,177.216,16.037,151.974
C08721=1099.337,151.308,-64.525,177.214,16.038,151.974
C08722=1099.332,151.059,-64.504,177.210,16.037,151.975
C08723=1099.326,150.810,-64.483,177.207,16.037,151.976
C08724=1099.320,150.561,-64.462,177.204,16.038,151.976
C08725=1099.315,150.312,-64.441,177.200,16.038,151.977
C08726=1099.309,150.063,-64.420,177.197,16.037,151.978
C08727=1099.303,149.814,-64.399,177.194,16.038,151.978
C08728=1099.298,149.564,-64.378,177.191,16.038,151.979
C08729=1099.293,149.316,-64.357,177.187,16.037,151.980
C08730=1099.287,149.067,-64.337,177.185,16.038,151.981
C08731=1099.281,148.817,-64.316,177.181,16.038,151.981
C08732=1099.275,148.569,-64.295,177.178,16.038,151.982
C08733=1099.270,148.320,-64.274,177.175,16.038,151.983
C08734=1099.264,148.070,-64.253,177.172,16.038,151.983
C08735=1099.259,147.821,-64.232,177.168,16.038,151.984
C08736=1099.253,147.573,-64.212,177.166,16.038,151.985
C08737=1099.247,147.323,-64.192,177.162,16.038,151.985
C08738=1099.241,147.074,-64.171,177.158,16.038,151.986
C08739=1099.236,146.825,-64.149,177.156,16.039,151.987
C08740=1099.230,146.576,-64.130,177.152,16.039,151.987
C08741=1099.225,146.327,-64.109,177.149,16.039,151.988
C08742=1099.219,146.077,-64.088,177.146,16.039,151.989
C08743=1099.213,145.829,-64.067,177.143,16.039,151.989
C08744=1099.207,145.580,-64.047,177.139,16.039,151.990
C08745=1099.202,145.331,-64.026,177.137,16.039,151.991
C08746=1099.196,145.081,-64.005,177.133,16.039,151.991
C08747=1099.191,144.832,-63.985,177.130,16.038,151.992
C08748=1099.185,144.583,-63.965,177.127,16.039,151.993
C08749=1099.179,144.310,-63.941,177.124,16.039,151.993
C08750=1099.172,144.036,-63.919,177.120,16.039,151.994
C08751=1099.166,143.762,-63.897,177.116,16.039,151.995
C08752=1099.160,143.487,-63.874,177.113,16.039,151.996
C08753=1099.154,143.239,-63.854,177.110,16.039,151.996
C08754=1099.149,142.989,-63.833,177.107,16.039,151.997
C08755=1099.143,142.740,-63.812,177.104,16.039,151.997
C08756=1099.138,142.490,-63.792,177.101,16.040,151.998
C08757=1099.132,142.242,-63.772,177.098,16.039,151.999
C08758=1099.127,141.992,-63.751,177.094,16.039,152.000
C08759=1099.121,141.743,-63.731,177.092,16.039,152.000
C08760=1099.115,141.494,-63.710,177.088,16.039,152.001
C08761=1099.109,141.245,-63.689,177.085,16.039,152.001
C08762=1099.104,140.996,-63.669,177.082,16.039,152.002
C08763=1099.098,140.747,-63.649,177.079,16.039,152.003
C08764=1099.093,140.498,-63.628,177.075,16.039,152.003
C08765=1099.087,140.249,-63.609,177.073,16.039,152.004
C08766=1099.082,140.000,-63.588,177.069,16.039,152.005
C08767=1099.075,139.750,-63.568,177.066,16.039,152.005
C08768=1099.070,139.501,-63.547,177.063,16.039,152.006
C08769=1099.065,139.252,-63.527,177.060,16.039,152.007
C08770=1099.059,139.003,-63.507,177.057,16.039,152.007
C08771=1099.054,138.754,-63.486,177.054,16.039,152.008
C08772=1099.048,138.505,-63.466,177.050,16.039,152.008
C08773=1099.042,138.256,-63.446,177.048,16.039,152.009
C08774=1099.036,138.007,-63.426,177.044,16.039,152.010
C08775=1099.031,137.758,-63.405,177.041,16.038,152.010
C08776=1099.024,137.509,-63.385,177.038,16.039,152.011
C08777=1099.019,137.259,-63.365,177.035,16.039,152.012
C08778=1099.013,137.010,-63.345,177.032,16.039,152.012
C08779=1099.008,136.761,-63.325,177.029,16.039,152.013
C08780=1099.002,136.512,-63.305,177.026,16.038,152.013
C08781=1098.996,136.263,-63.285,177.023,16.039,152.014
C08782=1098.991,136.014,-63.264,177.020,16.039,152.015
C08783=1098.985,135.765,-63.245,177.017,16.038,152.015
C08784=1098.980,135.516,-63.224,177.014,16.039,152.016
C08785=1098.974,135.267,-63.204,177.010,16.038,152.017
C08786=1098.969,135.018,-63.184,177.007,16.038,152.017
C08787=1098.963,134.769,-63.164,177.004,16.039,152.018
C08788=1098.958,134.519,-63.144,177.001,16.038,152.019
C08789=1098.951,134.270,-63.124,176.999,16.038,152.019
C08790=1098.945,134.021,-63.104,176.995,16.038,152.020
C08791=1098.940,133.771,-63.084,176.992,16.038,152.020
C08792=1098.934,133.522,-63.064,176.989,16.038,152.021
C08793=1098.929,133.273,-63.043,176.986,16.038,152.022
C08794=1098.923,133.024,-63.024,176.983,16.038,152.022
C08795=1098.917,132.775,-63.004,176.980,16.038,152.023
C08796=1098.912,132.526,-62.984,176.977,16.037,152.023
C08797=1098.906,132.277,-62.964,176.974,16.038,152.024
C08798=1098.900,132.028,-62.945,176.971,16.038,152.025
C08799=1098.895,131.778,-62.924,176.968,16.037,152.025
C08800=1098.890,131.529,-62.905,176.965,16.037,152.026
C08801=1098.884,131.280,-62.885,176.962,16.037,152.026
C08802=1098.878,131.031,-62.865,176.959,16.038,152.027
C08803=1098.873,130.782,-62.845,176.956,16.037,152.028
C08804=1098.867,130.533,-62.825,176.952,16.037,152.028
C08805=1098.861,130.283,-62.806,176.950,16.037,152.029
C08806=1098.855,130.035,-62.786,176.946,16.037,152.030
C08807=1098.849,129.786,-62.766,176.944,16.037,152.030
C08808=1098.844,129.536,-62.746,176.941,16.037,152.031
C08809=1098.838,129.287,-62.726,176.937,16.036,152.031
C08810=1098.832,129.038,-62.707,176.935,16.037,152.032
C08811=1098.826,128.789,-62.687,176.931,16.037,152.033
C08812=1098.821,128.540,-62.668,176.928,16.036,152.033
C08813=1098.816,128.325,-62.650,176.926,16.036,152.034
C08814=1098.811,128.110,-62.633,176.923,16.036,152.034
C08815=1098.806,127.895,-62.616,176.921,16.036,152.035
C08816=1098.801,127.681,-62.599,176.919,16.036,152.035
C08817=1098.797,127.465,-62.583,176.915,16.036,152.036
C08818=1098.792,127.251,-62.566,176.913,16.036,152.036
C08819=1098.786,127.036,-62.549,176.911,16.036,152.037
C08820=1098.781,126.820,-62.531,176.908,16.036,152.037
C08821=1098.776,126.572,-62.512,176.905,16.036,152.038
C08822=1098.770,126.323,-62.492,176.902,16.035,152.038
C08823=1098.765,126.074,-62.473,176.899,16.035,152.039
C08824=1098.759,125.825,-62.453,176.896,16.035,152.040
C08825=1098.753,125.575,-62.434,176.893,16.035,152.040
C08826=1098.747,125.326,-62.415,176.890,16.035,152.041
C08827=1098.741,125.077,-62.395,176.887,16.034,152.041
C08828=1098.736,124.827,-62.375,176.884,16.034,152.042
C08829=1098.731,124.578,-62.356,176.881,16.034,152.042
C08830=1098.725,124.329,-62.336,176.879,16.034,152.043
C08831=1098.719,124.080,-62.316,176.875,16.034,152.044
C08832=1098.714,123.831,-62.298,176.872,16.033,152.044
C08833=1098.708,123.582,-62.278,176.870,16.034,152.045
C08834=1098.702,123.333,-62.258,176.866,16.033,152.045
C08835=1098.697,123.083,-62.239,176.864,16.033,152.046
C08836=1098.691,122.834,-62.219,176.861,16.033,152.046
C08837=1098.685,122.585,-62.200,176.857,16.033,152.047
C08838=1098.679,122.336,-62.181,176.855,16.033,152.048
C08839=1098.674,122.087,-62.162,176.852,16.032,152.048
C08840=1098.668,121.838,-62.142,176.849,16.032,152.049
C08841=1098.662,121.589,-62.123,176.846,16.032,152.049
C08842=1098.657,121.339,-62.103,176.843,16.032,152.050
C08843=1098.652,121.089,-62.083,176.840,16.032,152.050
C08844=1098.646,120.840,-62.064,176.837,16.031,152.051
C08845=1098.641,120.592,-62.045,176.834,16.032,152.052
C08846=1098.635,120.342,-62.025,176.831,16.031,152.052
C08847=1098.629,120.093,-62.006,176.828,16.030,152.053
C08848=1098.624,119.844,-61.987,176.826,16.030,152.053
C08849=1098.618,119.594,-61.968,176.822,16.030,152.054
C08850=1098.613,119.345,-61.949,176.820,16.030,152.054
C08851=1098.607,119.097,-61.929,176.817,16.030,152.055
C08852=1098.601,118.847,-61.910,176.813,16.029,152.055
C08853=1098.595,118.598,-61.890,176.811,16.030,152.056
C08854=1098.590,118.349,-61.871,176.808,16.029,152.056
C08855=1098.585,118.100,-61.852,176.805,16.029,152.057
C08856=1098.579,117.850,-61.833,176.802,16.029,152.058
C08857=1098.573,117.601,-61.814,176.800,16.029,152.058
C08858=1098.568,117.352,-61.795,176.797,16.028,152.059
C08859=1098.562,117.103,-61.776,176.793,16.027,152.059
C08860=1098.556,116.853,-61.757,176.791,16.028,152.060
C08861=1098.551,116.605,-61.738,176.788,16.027,152.060
C08862=1098.545,116.355,-61.719,176.786,16.027,152.061
C08863=1098.540,116.106,-61.700,176.782,16.027,152.061
C08864=1098.534,115.856,-61.680,176.779,16.026,152.062
C08865=1098.526,115.514,-61.654,176.775,16.026,152.063
C08866=1098.519,115.171,-61.628,176.771,16.025,152.063
C08867=1098.512,114.828,-61.602,176.768,16.025,152.064
C08868=1098.504,114.486,-61.576,176.763,16.025,152.065
C08869=1098.498,114.236,-61.556,176.761,16.025,152.065
C08870=1098.493,113.987,-61.537,176.758,16.024,152.066
C08871=1098.486,113.738,-61.518,176.756,16.024,152.066
C08872=1098.481,113.489,-61.500,176.752,16.024,152.067
C08873=1098.475,113.239,-61.480,176.749,16.023,152.067
C08874=1098.470,112.990,-61.461,176.747,16.023,152.068
C08875=1098.464,112.742,-61.443,176.744,16.023,152.068
C08876=1098.459,112.491,-61.424,176.741,16.023,152.069
C08877=1098.452,112.217,-61.403,176.738,16.022,152.070
C08878=1098.446,111.943,-61.382,176.735,16.022,152.070
C08879=1098.439,111.669,-61.361,176.732,16.021,152.071
C08880=1098.434,111.395,-61.341,176.728,16.021,152.071
C08881=1098.428,111.145,-61.322,176.726,16.021,152.072
C08882=1098.423,110.897,-61.303,176.723,16.021,152.072
C08883=1098.417,110.647,-61.284,176.720,16.020,152.073
C08884=1098.411,110.398,-61.266,176.717,16.020,152.073
C08885=1098.406,110.149,-61.247,176.715,16.020,152.074
C08886=1098.399,109.900,-61.228,176.712,16.019,152.074
C08887=1098.394,109.650,-61.209,176.709,16.019,152.075
C08888=1098.388,109.401,-61.190,176.706,16.019,152.076
C08889=1098.382,109.152,-61.172,176.703,16.018,152.076
C08890=1098.377,108.902,-61.153,176.700,16.018,152.076
C08891=1098.372,108.654,-61.134,176.697,16.018,152.077
C08892=1098.366,108.404,-61.116,176.695,16.018,152.077
C08893=1098.360,108.154,-61.097,176.692,16.017,152.078
C08894=1098.354,107.906,-61.079,176.690,16.017,152.078
C08895=1098.348,107.657,-61.060,176.686,16.017,152.079
C08896=1098.343,107.407,-61.041,176.684,16.016,152.079
C08897=1098.337,107.158,-61.023,176.681,16.016,152.080
C08898=1098.331,106.909,-61.004,176.678,16.016,152.081
C08899=1098.326,106.660,-60.986,176.675,16.015,152.081
C08900=1098.320,106.410,-60.967,176.672,16.015,152.082
C08901=1098.315,106.161,-60.948,176.670,16.015,152.082
C08902=1098.309,105.912,-60.930,176.667,16.014,152.083
C08903=1098.303,105.662,-60.911,176.664,16.014,152.083
C08904=1098.298,105.413,-60.893,176.661,16.014,152.084
C08905=1098.292,105.164,-60.874,176.659,16.013,152.084
C08906=1098.286,104.915,-60.855,176.656,16.013,152.085
C08907=1098.281,104.665,-60.837,176.653,16.012,152.085
C08908=1098.275,104.416,-60.818,176.650,16.012,152.086
C08909=1098.270,104.167,-60.800,176.647,16.011,152.086
C08910=1098.263,103.918,-60.782,176.645,16.011,152.086
C08911=1098.259,103.668,-60.763,176.642,16.011,152.087
C08912=1098.253,103.419,-60.744,176.640,16.010,152.087
C08913=1098.247,103.170,-60.727,176.636,16.010,152.088
C08914=1098.242,102.921,-60.707,176.634,16.010,152.088
C08915=1098.236,102.671,-60.690,176.631,16.009,152.089
C08916=1098.230,102.422,-60.671,176.629,16.009,152.089
C08917=1098.225,102.173,-60.653,176.626,16.008,152.090
C08918=1098.219,101.924,-60.634,176.623,16.008,152.090
C08919=1098.214,101.675,-60.616,176.620,16.008,152.091
C08920=1098.208,101.425,-60.597,176.617,16.007,152.091
C08921=1098.202,101.176,-60.579,176.615,16.007,152.092
C08922=1098.196,100.926,-60.561,176.612,16.006,152.092
C08923=1098.191,100.677,-60.542,176.609,16.006,152.093
C08924=1098.185,100.428,-60.525,176.607,16.005,152.093
C08925=1098.179,100.179,-60.506,176.604,16.005,152.094
C08926=1098.174,99.929,-60.488,176.601,16.005,152.094
C08927=1098.168,99.680,-60.469,176.599,16.005,152.095
C08928=1098.162,99.431,-60.452,176.596,16.004,152.095
C08929=1098.157,99.181,-60.433,176.593,16.004,152.096
C08930=1098.151,98.933,-60.415,176.590,16.003,152.096
C08931=1098.145,98.683,-60.397,176.588,16.003,152.097
C08932=1098.140,98.434,-60.379,176.585,16.002,152.097
C08933=1098.133,98.185,-60.360,176.582,16.001,152.097
C08934=1098.128,97.935,-60.343,176.580,16.002,152.098
C08935=1098.123,97.685,-60.324,176.577,16.001,152.098
C08936=1098.117,97.437,-60.306,176.574,16.001,152.099
C08937=1098.111,97.187,-60.288,176.571,16.000,152.099
C08938=1098.106,96.938,-60.270,176.569,16.000,152.100
C08939=1098.100,96.689,-60.252,176.566,15.999,152.100
C08940=1098.094,96.440,-60.233,176.564,15.999,152.101
C08941=1098.088,96.166,-60.214,176.561,15.998,152.101
C08942=1098.082,95.891,-60.194,176.558,15.998,152.102
C08943=1098.075,95.618,-60.174,176.554,15.997,152.102
C08944=1098.069,95.343,-60.154,176.552,15.997,152.103
C08945=1098.063,95.094,-60.137,176.549,15.997,152.103
C08946=1098.058,94.845,-60.118,176.547,15.996,152.104
C08947=1098.052,94.595,-60.100,176.544,15.995,152.104
C08948=1098.047,94.346,-60.082,176.542,15.995,152.104
C08949=1098.041,94.097,-60.065,176.539,15.994,152.105
C08950=1098.036,93.847,-60.046,176.536,15.995,152.105
C08951=1098.030,93.598,-60.029,176.533,15.994,152.106
C08952=1098.024,93.349,-60.010,176.531,15.993,152.106
C08953=1098.018,93.100,-59.992,176.528,15.993,152.107
C08954=1098.013,92.850,-59.974,176.525,15.992,152.107
C08955=1098.007,92.601,-59.956,176.523,15.991,152.108
C08956=1098.002,92.352,-59.939,176.519,15.991,152.108
C08957=1097.996,92.103,-59.921,176.517,15.991,152.109
C08958=1097.990,91.853,-59.903,176.514,15.990,152.109
C08959=1097.985,91.604,-59.885,176.512,15.990,152.109
C08960=1097.979,91.354,-59.867,176.509,15.989,152.110
C08961=1097.974,91.105,-59.849,176.507,15.989,152.110
C08962=1097.968,90.856,-59.832,176.504,15.988,152.111
C08963=1097.962,90.606,-59.814,176.502,15.987,152.111
C08964=1097.956,90.358,-59.796,176.499,15.987,152.112
C08965=1097.951,90.108,-59.778,176.496,15.987,152.112
C08966=1097.945,89.859,-59.760,176.493,15.986,152.113
C08967=1097.939,89.610,-59.743,176.491,15.986,152.113
C08968=1097.933,89.360,-59.725,176.488,15.985,152.113
C08969=1097.927,89.111,-59.707,176.486,15.985,152.114
C08970=1097.922,88.862,-59.690,176.483,15.984,152.114
C08971=1097.916,88.612,-59.672,176.481,15.983,152.115
C08972=1097.910,88.363,-59.654,176.478,15.983,152.115
C08973=1097.905,88.114,-59.637,176.475,15.983,152.116
C08974=1097.899,87.864,-59.619,176.473,15.982,152.116
C08975=1097.893,87.615,-59.602,176.470,15.982,152.116
C08976=1097.888,87.366,-59.584,176.467,15.981,152.117
C08977=1097.882,87.116,-59.566,176.465,15.981,152.117
C08978=1097.876,86.867,-59.549,176.462,15.980,152.118
C08979=1097.871,86.618,-59.531,176.460,15.980,152.118
C08980=1097.865,86.368,-59.513,176.457,15.979,152.119
C08981=1097.859,86.119,-59.496,176.455,15.978,152.119
C08982=1097.854,85.870,-59.478,176.452,15.978,152.119
C08983=1097.848,85.621,-59.460,176.450,15.977,152.120
C08984=1097.842,85.371,-59.443,176.447,15.976,152.120
C08985=1097.837,85.122,-59.426,176.445,15.976,152.121
C08986=1097.831,84.872,-59.408,176.442,15.975,152.121
C08987=1097.825,84.623,-59.390,176.439,15.975,152.121
C08988=1097.820,84.374,-59.373,176.436,15.974,152.122
C08989=1097.814,84.125,-59.355,176.434,15.974,152.122
C08990=1097.809,83.875,-59.338,176.431,15.973,152.123
C08991=1097.803,83.625,-59.320,176.429,15.973,152.123
C08992=1097.797,83.376,-59.303,176.426,15.972,152.124
C08993=1097.792,83.127,-59.285,176.424,15.972,152.124
C08994=1097.786,82.878,-59.268,176.421,15.971,152.124
C08995=1097.780,82.628,-59.250,176.419,15.971,152.125
C08996=1097.775,82.379,-59.233,176.417,15.970,152.125
C08997=1097.769,82.130,-59.216,176.414,15.969,152.125
C08998=1097.763,81.880,-59.199,176.412,15.969,152.126
C08999=1097.758,81.631,-59.181,176.409,15.968,152.126
C09000=1097.752,81.382,-59.163,176.407,15.968,152.127
C09001=1097.747,81.132,-59.147,176.404,15.967,152.127
C09002=1097.741,80.883,-59.129,176.401,15.967,152.128
C09003=1097.735,80.634,-59.111,176.398,15.966,152.128
C09004=1097.730,80.385,-59.094,176.397,15.965,152.128
C09005=1097.724,80.110,-59.075,176.394,15.964,152.129
C09006=1097.717,79.836,-59.056,176.391,15.963,152.129
C09007=1097.711,79.562,-59.037,176.388,15.963,152.130
C09008=1097.705,79.288,-59.018,176.385,15.962,152.130
C09009=1097.699,79.038,-59.001,176.382,15.961,152.130
C09010=1097.693,78.789,-58.984,176.380,15.961,152.131
C09011=1097.688,78.540,-58.967,176.377,15.960,152.131
C09012=1097.682,78.291,-58.949,176.375,15.960,152.132
C09013=1097.677,78.042,-58.932,176.372,15.959,152.132
C09014=1097.672,77.792,-58.915,176.370,15.959,152.132
C09015=1097.665,77.543,-58.898,176.367,15.958,152.133
C09016=1097.660,77.293,-58.881,176.365,15.957,152.133
C09017=1097.654,77.044,-58.863,176.362,15.957,152.134
C09018=1097.648,76.794,-58.847,176.360,15.956,152.134
C09019=1097.643,76.545,-58.829,176.358,15.956,152.134
C09020=1097.637,76.296,-58.813,176.355,15.955,152.135
C09021=1097.631,76.046,-58.795,176.353,15.955,152.135
C09022=1097.625,75.797,-58.778,176.350,15.954,152.136
C09023=1097.620,75.548,-58.761,176.348,15.953,152.136
C09024=1097.614,75.298,-58.745,176.345,15.952,152.136
C09025=1097.608,75.049,-58.727,176.343,15.952,152.137
C09026=1097.603,74.800,-58.710,176.340,15.951,152.137
C09027=1097.597,74.551,-58.693,176.338,15.951,152.137
C09028=1097.591,74.301,-58.676,176.335,15.950,152.138
C09029=1097.586,74.051,-58.658,176.333,15.949,152.138
C09030=1097.580,73.802,-58.642,176.330,15.948,152.139
C09031=1097.574,73.553,-58.625,176.328,15.948,152.139
C09032=1097.569,73.303,-58.608,176.325,15.947,152.139
C09033=1097.563,73.054,-58.591,176.323,15.947,152.140
C09034=1097.557,72.805,-58.574,176.321,15.946,152.140
C09035=1097.552,72.555,-58.557,176.318,15.945,152.140
C09036=1097.546,72.307,-58.540,176.316,15.945,152.141
C09037=1097.541,72.057,-58.523,176.313,15.944,152.141
C09038=1097.534,71.807,-58.507,176.311,15.943,152.141
C09039=1097.529,71.558,-58.489,176.308,15.942,152.142
C09040=1097.523,71.308,-58.472,176.306,15.942,152.142
C09041=1097.517,71.059,-58.456,176.303,15.941,152.143
C09042=1097.512,70.810,-58.438,176.301,15.941,152.143
C09043=1097.506,70.561,-58.422,176.298,15.939,152.143
C09044=1097.501,70.311,-58.405,176.296,15.939,152.144
C09045=1097.495,70.062,-58.388,176.294,15.939,152.144
C09046=1097.489,69.812,-58.371,176.291,15.937,152.144
C09047=1097.483,69.563,-58.355,176.289,15.937,152.145
C09048=1097.478,69.314,-58.338,176.286,15.936,152.145
C09049=1097.472,69.065,-58.321,176.284,15.936,152.145
C09050=1097.467,68.815,-58.304,176.281,15.935,152.146
C09051=1097.461,68.566,-58.288,176.279,15.935,152.146
C09052=1097.455,68.317,-58.271,176.276,15.933,152.147
C09053=1097.449,68.067,-58.254,176.274,15.933,152.147
C09054=1097.444,67.818,-58.238,176.272,15.932,152.147
C09055=1097.438,67.568,-58.221,176.269,15.932,152.148
C09056=1097.433,67.319,-58.204,176.267,15.931,152.148
C09057=1097.427,67.070,-58.187,176.264,15.930,152.148
C09058=1097.421,66.820,-58.171,176.262,15.930,152.149
C09059=1097.415,66.571,-58.154,176.260,15.928,152.149
C09060=1097.410,66.321,-58.137,176.257,15.928,152.149
C09061=1097.404,66.072,-58.121,176.255,15.927,152.150
C09062=1097.398,65.823,-58.105,176.253,15.927,152.150
C09063=1097.393,65.574,-58.087,176.251,15.926,152.150
C09064=1097.387,65.324,-58.071,176.248,15.925,152.151
C09065=1097.382,65.075,-58.054,176.245,15.925,152.151
C09066=1097.376,64.825,-58.038,176.243,15.923,152.151
C09067=1097.370,64.576,-58.022,176.241,15.923,152.152
C09068=1097.365,64.326,-58.005,176.238,15.922,152.152
